// TIA Portal V20 export
FUNCTION_BLOCK "Sequence_2_TransferPnPRight"   // FB32855, LAD
TITLE = Sequence
// Sequence template programmend in ladder logic
// stored: IsIECCheckEnabled true, MemoryReserve 100, Namespace Unit1.Em5, SetENOAutomatically true
   VAR_INPUT
      unitStatus { ExternalAccessible := 'False'; ExternalVisible := 'False'; ExternalWritable := 'False'} : "LAF_typeUnitStatus";
   END_VAR
   VAR
      instSequenceLADControl { ExternalAccessible := 'False'; ExternalVisible := 'False'; ExternalWritable := 'False'} : "LAF_ControlLadSequence";
      instSequenceLADStatus { ExternalAccessible := 'False'; ExternalVisible := 'False'; ExternalWritable := 'False'} : "LAF_StatusLadSequence";
      statTonTime { ExternalAccessible := 'False'; ExternalVisible := 'False'; ExternalWritable := 'False'} : Array[0..9999] of TON_TIME;
      NoDataCheck { S7_SetPoint := 'True'} : "LER_typePartData";
   END_VAR
   VAR_TEMP
      tempCustomerAction : Bool;   // Placeholder for possible actions
      tempDo_nothing_and_wait_for_init : Bool;   // Placeholder for doing nothing
      tempSafeStateCondition : Bool;   // Temp Condition for the equipment module to be in a safe state
   END_VAR
   VAR CONSTANT
      delayTime : Time := T#500ms;
      STEP_IDLE : DInt := 1;
      JOB_1_STEP_01 : DInt := 101;
      JOB_1_STEP_10 : DInt := 110;
      JOB_1_STEP_20 : DInt := 120;
      JOB_1_STEP_30 : DInt := 130;
      JOB_1_STEP_40 : DInt := 140;
      JOB_1_STEP_50 : DInt := 150;
      JOB_1_STEP_60 : DInt := 160;
      JOB_1_STEP_70 : DInt := 170;
      JOB_1_STEP_80 : DInt := 180;
      JOB_1_STEP_90 : DInt := 190;
      JOB_2_STEP_01 : DInt := 201;
      JOB_2_STEP_10 : DInt := 210;
      JOB_2_STEP_20 : DInt := 220;
      JOB_2_STEP_30 : DInt := 230;
      JOB_2_STEP_40 : DInt := 240;
      JOB_2_STEP_80 : DInt := 280;
      JOB_2_STEP_81 : DInt := 281;
      JOB_2_STEP_90 : DInt := 290;
      JOB_3_STEP_01 : DInt := 301;
      JOB_3_STEP_10 : DInt := 310;
      JOB_3_STEP_20 : DInt := 320;
      JOB_3_STEP_30 : DInt := 330;
      JOB_3_STEP_40 : DInt := 340;
      JOB_3_STEP_50 : DInt := 350;
      JOB_3_STEP_80 : DInt := 380;
      JOB_3_STEP_81 : DInt := 381;
      JOB_3_STEP_90 : DInt := 390;
      JOB_4_STEP_01 : DInt := 401;
      JOB_4_STEP_10 : DInt := 410;
      JOB_4_STEP_20 : DInt := 420;
      JOB_4_STEP_30 : DInt := 430;
      JOB_4_STEP_40 : DInt := 440;
      JOB_4_STEP_80 : DInt := 480;
      JOB_4_STEP_81 : DInt := 481;
      JOB_4_STEP_90 : DInt := 490;
      JOB_5_STEP_01 : DInt := 501;
      JOB_5_STEP_10 : DInt := 510;
      JOB_5_STEP_20 : DInt := 520;
      JOB_5_STEP_30 : DInt := 530;
      JOB_5_STEP_40 : DInt := 540;
      JOB_5_STEP_50 : DInt := 550;
      JOB_5_STEP_80 : DInt := 580;
      JOB_5_STEP_81 : DInt := 581;
      JOB_5_STEP_90 : DInt := 590;
      JOB_6_STEP_01 : DInt := 601;
      JOB_6_STEP_10 : DInt := 610;
      JOB_6_STEP_20 : DInt := 620;
      JOB_6_STEP_30 : DInt := 630;
      JOB_6_STEP_40 : DInt := 640;
      JOB_6_STEP_50 : DInt := 650;
      JOB_6_STEP_51 : DInt := 651;
      JOB_6_STEP_52 : DInt := 652;
      JOB_6_STEP_80 : DInt := 680;
      JOB_6_STEP_81 : DInt := 681;
      JOB_6_STEP_90 : DInt := 690;
      JOB_7_STEP_01 : DInt := 701;
      JOB_7_STEP_10 : DInt := 710;
      JOB_7_STEP_20 : DInt := 720;
      JOB_7_STEP_30 : DInt := 730;
      JOB_7_STEP_40 : DInt := 740;
      JOB_7_STEP_50 : DInt := 750;
      JOB_7_STEP_80 : DInt := 780;
      JOB_7_STEP_81 : DInt := 781;
      JOB_7_STEP_90 : DInt := 790;
      JOB_8_STEP_01 : DInt := 801;
      JOB_8_STEP_10 : DInt := 810;
      JOB_8_STEP_20 : DInt := 820;
      JOB_8_STEP_30 : DInt := 830;
      JOB_8_STEP_40 : DInt := 840;
      JOB_8_STEP_50 : DInt := 850;
      JOB_8_STEP_51 : DInt := 851;
      JOB_8_STEP_52 : DInt := 852;
      JOB_8_STEP_80 : DInt := 880;
      JOB_8_STEP_81 : DInt := 881;
      JOB_8_STEP_90 : DInt := 890;
      JOB_9_STEP_01 : DInt := 901;
      JOB_9_STEP_10 : DInt := 910;
      JOB_9_STEP_20 : DInt := 920;
      JOB_9_STEP_30 : DInt := 930;
      JOB_9_STEP_31 : DInt := 931;
      JOB_9_STEP_40 : DInt := 940;
      JOB_9_STEP_50 : DInt := 950;
      JOB_9_STEP_80 : DInt := 980;
      JOB_9_STEP_81 : DInt := 981;
      JOB_9_STEP_82 : DInt := 982;
      JOB_9_STEP_90 : DInt := 990;
      STEP_IMMEDIATE_STOP : DInt := 9001;   // Step executed when an immediate stop command is triggered for the sequence (i.e. when unit is in state aborting)
      TO_DO_INSERT_ACTIONS_HERE : Bool := TRUE;   // Template : Add actions
      TO_DO_INSERT_CONDITION_FOR_TRANSITION_HERE : Bool := TRUE;   // Template : Add conditions
   END_VAR
   VAR_TEMP   // added for the SCL form of the ladder/FBD networks
      _w1 : Bool;
      _w2 : Bool;
      _w3 : Bool;
      _w4 : Bool;
      _w5 : Bool;
      _w6 : Bool;
   END_VAR
BEGIN

REGION Network 1: BLOCK INFO HEADER
   // (company) / (C) Copyright (year)
   // ---------------------------------------------------------------------------------
   // Title:                             (Title of this block)
   // Comment/Function: (that is implemented in the block)
   // Library/Family:           (that the source is dedicated to)
   // Author:                        (department / person in charge / contact)
   // Target System:          (test system with FW version)
   // Engineering:              TIA Portal (SW version)
   // Restrictions:               (OB types, etc.)
   // Requirements:           (hardware, technological package, etc.)
   // ---------------------------------------------------------------------------------
   // Change log table:
   // Version          | Date             | Signature      | Expert in charge  | Changes applied ------------------------|----------------------|-------------------------|--------------------------------|-----------------------
   // 001.000.000 | yyyy-mm-dd | 0x00000000 | (name of expert) | First released version
END_REGION

REGION Network 2: DESCRIPTION
   // This is a template block provided by the Automation Framework. It can be used to create an own project.
   // The Block Info Header is prepared to put in your own data.
   // Description of the block could be added here and the docu created by Code2Docu.
END_REGION

REGION Network 3: ********************* CONTROL *************************
END_REGION

REGION Network 4: Sequence Control ("Enter your Sequins number here")
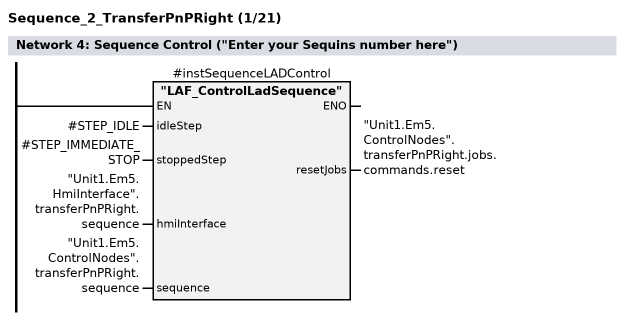
   RUNG wire#powerrail
      #instSequenceLADControl(idleStep := #STEP_IDLE, stoppedStep := #STEP_IMMEDIATE_STOP, hmiInterface := "Unit1.Em5.HmiInterface".transferPnPRight.sequence, sequence := "Unit1.Em5.ControlNodes".transferPnPRight.sequence, resetJobs => "Unit1.Em5.ControlNodes".transferPnPRight.jobs.commands.reset)
   END_RUNG
   // the same network as SCL:
   #instSequenceLADControl(idleStep := #STEP_IDLE,   // "LAF_ControlLadSequence"
                           stoppedStep := #STEP_IMMEDIATE_STOP,
                           hmiInterface := "Unit1.Em5.HmiInterface".transferPnPRight.sequence,
                           sequence := "Unit1.Em5.ControlNodes".transferPnPRight.sequence,
                           resetJobs => "Unit1.Em5.ControlNodes".transferPnPRight.jobs.commands.reset);
END_REGION

REGION Network 5: Step Idle
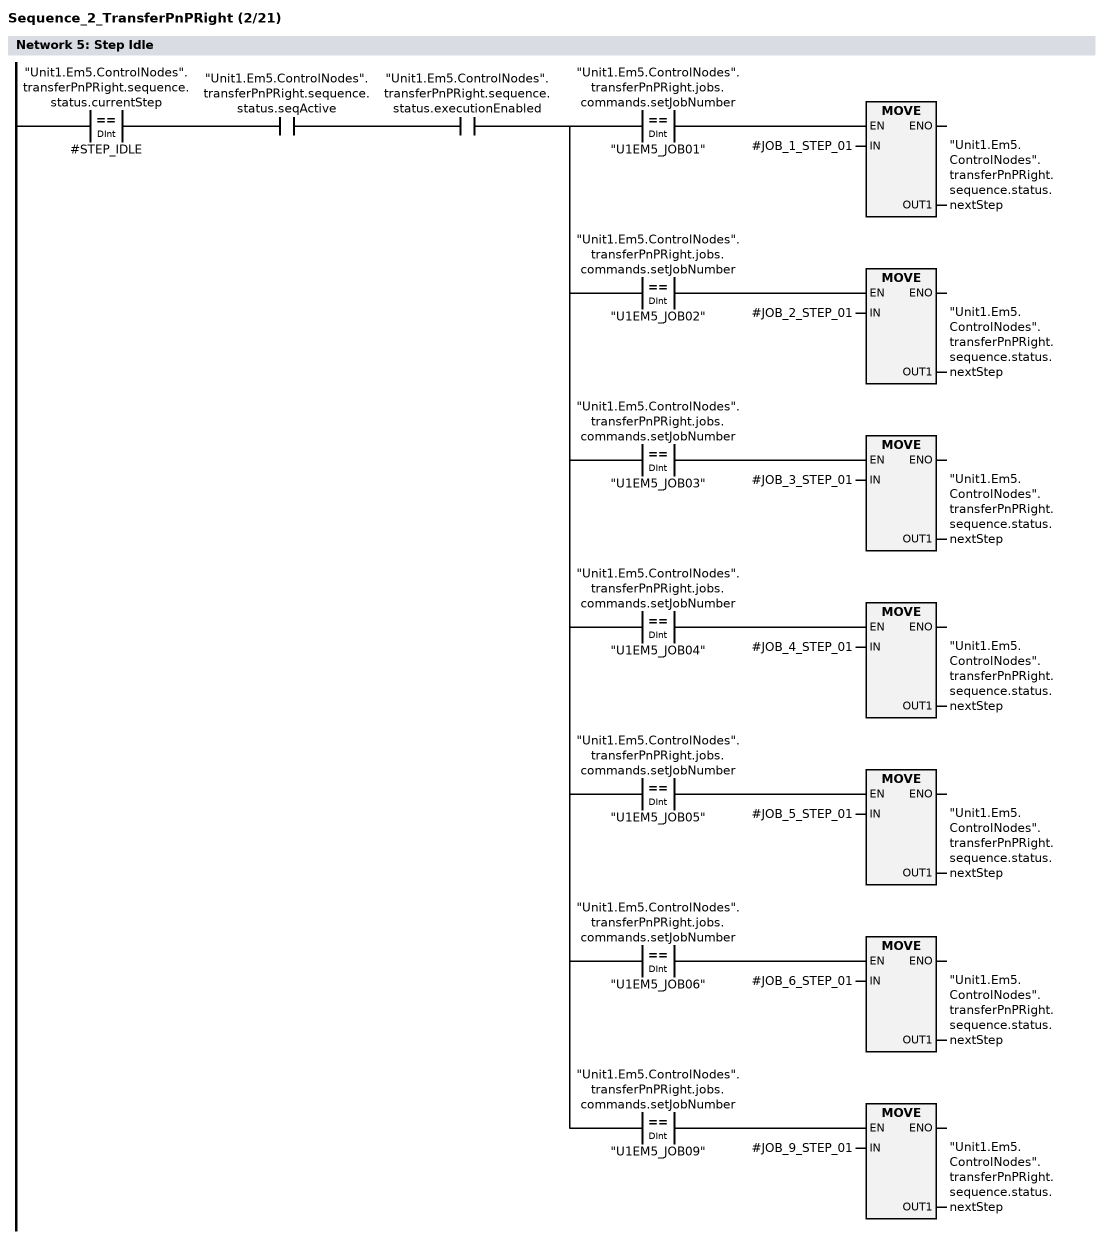
   RUNG wire#powerrail
      { S7_Templates := "SrcType := DInt" } EQ_Contact(in1 := "Unit1.Em5.ControlNodes".transferPnPRight.sequence.status.currentStep, in2 := #STEP_IDLE)
      Contact( "Unit1.Em5.ControlNodes".transferPnPRight.sequence.status.seqActive )
      Contact( "Unit1.Em5.ControlNodes".transferPnPRight.sequence.status.executionEnabled )
      wire#w1
      { S7_Templates := "SrcType := DInt" } EQ_Contact(in1 := "Unit1.Em5.ControlNodes".transferPnPRight.jobs.commands.setJobNumber, in2 := "U1EM5_JOB01")
      Move(in := #JOB_1_STEP_01, out1 => "Unit1.Em5.ControlNodes".transferPnPRight.sequence.status.nextStep)
   END_RUNG
   RUNG wire#w1
      { S7_Templates := "SrcType := DInt" } EQ_Contact(in1 := "Unit1.Em5.ControlNodes".transferPnPRight.jobs.commands.setJobNumber, in2 := "U1EM5_JOB02")
      Move(in := #JOB_2_STEP_01, out1 => "Unit1.Em5.ControlNodes".transferPnPRight.sequence.status.nextStep)
   END_RUNG
   RUNG wire#w1
      { S7_Templates := "SrcType := DInt" } EQ_Contact(in1 := "Unit1.Em5.ControlNodes".transferPnPRight.jobs.commands.setJobNumber, in2 := "U1EM5_JOB03")
      Move(in := #JOB_3_STEP_01, out1 => "Unit1.Em5.ControlNodes".transferPnPRight.sequence.status.nextStep)
   END_RUNG
   RUNG wire#w1
      { S7_Templates := "SrcType := DInt" } EQ_Contact(in1 := "Unit1.Em5.ControlNodes".transferPnPRight.jobs.commands.setJobNumber, in2 := "U1EM5_JOB04")
      Move(in := #JOB_4_STEP_01, out1 => "Unit1.Em5.ControlNodes".transferPnPRight.sequence.status.nextStep)
   END_RUNG
   RUNG wire#w1
      { S7_Templates := "SrcType := DInt" } EQ_Contact(in1 := "Unit1.Em5.ControlNodes".transferPnPRight.jobs.commands.setJobNumber, in2 := "U1EM5_JOB05")
      Move(in := #JOB_5_STEP_01, out1 => "Unit1.Em5.ControlNodes".transferPnPRight.sequence.status.nextStep)
   END_RUNG
   RUNG wire#w1
      { S7_Templates := "SrcType := DInt" } EQ_Contact(in1 := "Unit1.Em5.ControlNodes".transferPnPRight.jobs.commands.setJobNumber, in2 := "U1EM5_JOB06")
      Move(in := #JOB_6_STEP_01, out1 => "Unit1.Em5.ControlNodes".transferPnPRight.sequence.status.nextStep)
   END_RUNG
   RUNG wire#w1
      { S7_Templates := "SrcType := DInt" } EQ_Contact(in1 := "Unit1.Em5.ControlNodes".transferPnPRight.jobs.commands.setJobNumber, in2 := "U1EM5_JOB09")
      Move(in := #JOB_9_STEP_01, out1 => "Unit1.Em5.ControlNodes".transferPnPRight.sequence.status.nextStep)
   END_RUNG
   // the same network as SCL:
   #_w1 := ("Unit1.Em5.ControlNodes".transferPnPRight.sequence.status.currentStep = #STEP_IDLE) AND "Unit1.Em5.ControlNodes".transferPnPRight.sequence.status.seqActive AND "Unit1.Em5.ControlNodes".transferPnPRight.sequence.status.executionEnabled;
   IF #_w1 AND ("Unit1.Em5.ControlNodes".transferPnPRight.jobs.commands.setJobNumber = "U1EM5_JOB01") THEN
       "Unit1.Em5.ControlNodes".transferPnPRight.sequence.status.nextStep := #JOB_1_STEP_01;
   END_IF;
   IF #_w1 AND ("Unit1.Em5.ControlNodes".transferPnPRight.jobs.commands.setJobNumber = "U1EM5_JOB02") THEN
       "Unit1.Em5.ControlNodes".transferPnPRight.sequence.status.nextStep := #JOB_2_STEP_01;
   END_IF;
   IF #_w1 AND ("Unit1.Em5.ControlNodes".transferPnPRight.jobs.commands.setJobNumber = "U1EM5_JOB03") THEN
       "Unit1.Em5.ControlNodes".transferPnPRight.sequence.status.nextStep := #JOB_3_STEP_01;
   END_IF;
   IF #_w1 AND ("Unit1.Em5.ControlNodes".transferPnPRight.jobs.commands.setJobNumber = "U1EM5_JOB04") THEN
       "Unit1.Em5.ControlNodes".transferPnPRight.sequence.status.nextStep := #JOB_4_STEP_01;
   END_IF;
   IF #_w1 AND ("Unit1.Em5.ControlNodes".transferPnPRight.jobs.commands.setJobNumber = "U1EM5_JOB05") THEN
       "Unit1.Em5.ControlNodes".transferPnPRight.sequence.status.nextStep := #JOB_5_STEP_01;
   END_IF;
   IF #_w1 AND ("Unit1.Em5.ControlNodes".transferPnPRight.jobs.commands.setJobNumber = "U1EM5_JOB06") THEN
       "Unit1.Em5.ControlNodes".transferPnPRight.sequence.status.nextStep := #JOB_6_STEP_01;
   END_IF;
   IF #_w1 AND ("Unit1.Em5.ControlNodes".transferPnPRight.jobs.commands.setJobNumber = "U1EM5_JOB09") THEN
       "Unit1.Em5.ControlNodes".transferPnPRight.sequence.status.nextStep := #JOB_9_STEP_01;
   END_IF;
END_REGION

REGION Network 6: *************** JOB[1] EM HOMING ************************
END_REGION

REGION Network 7: Step[101] : JOB[1] Condition
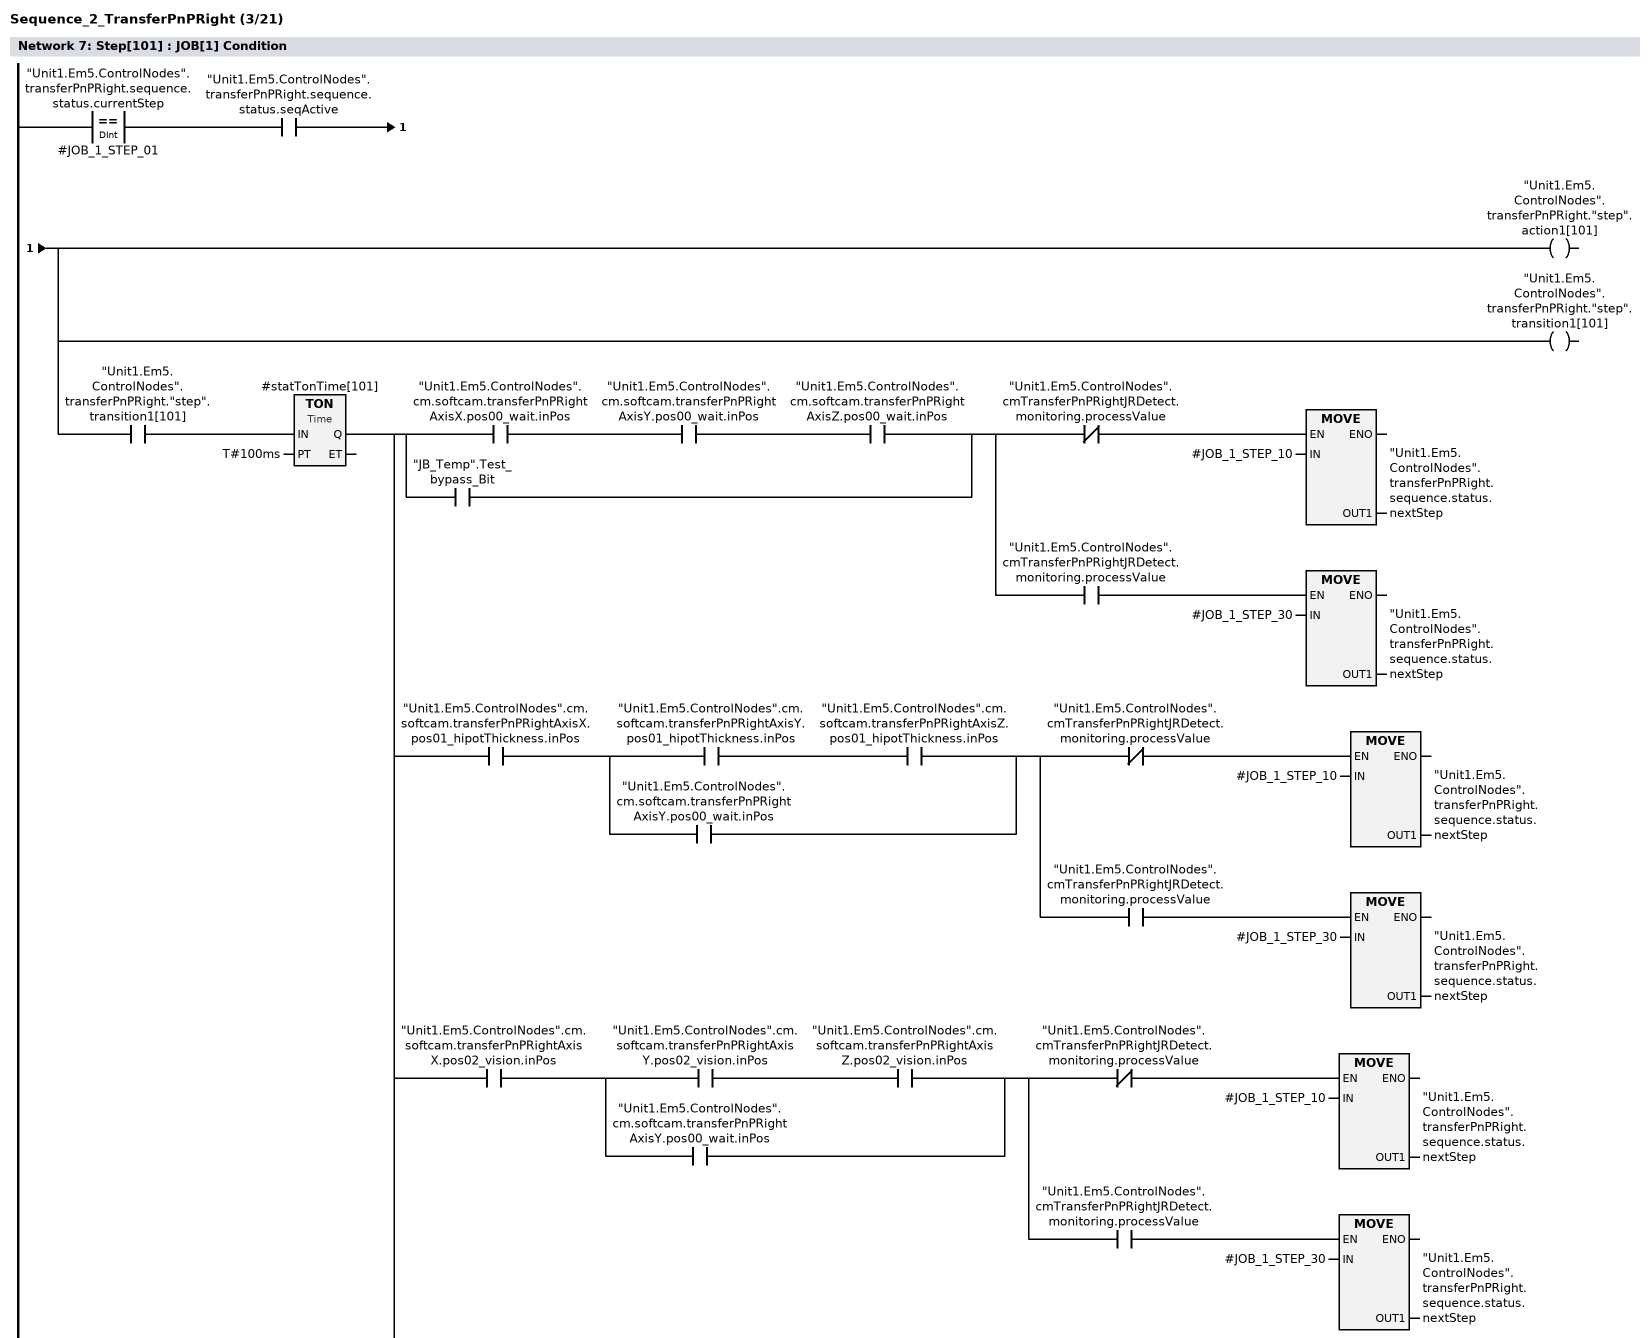
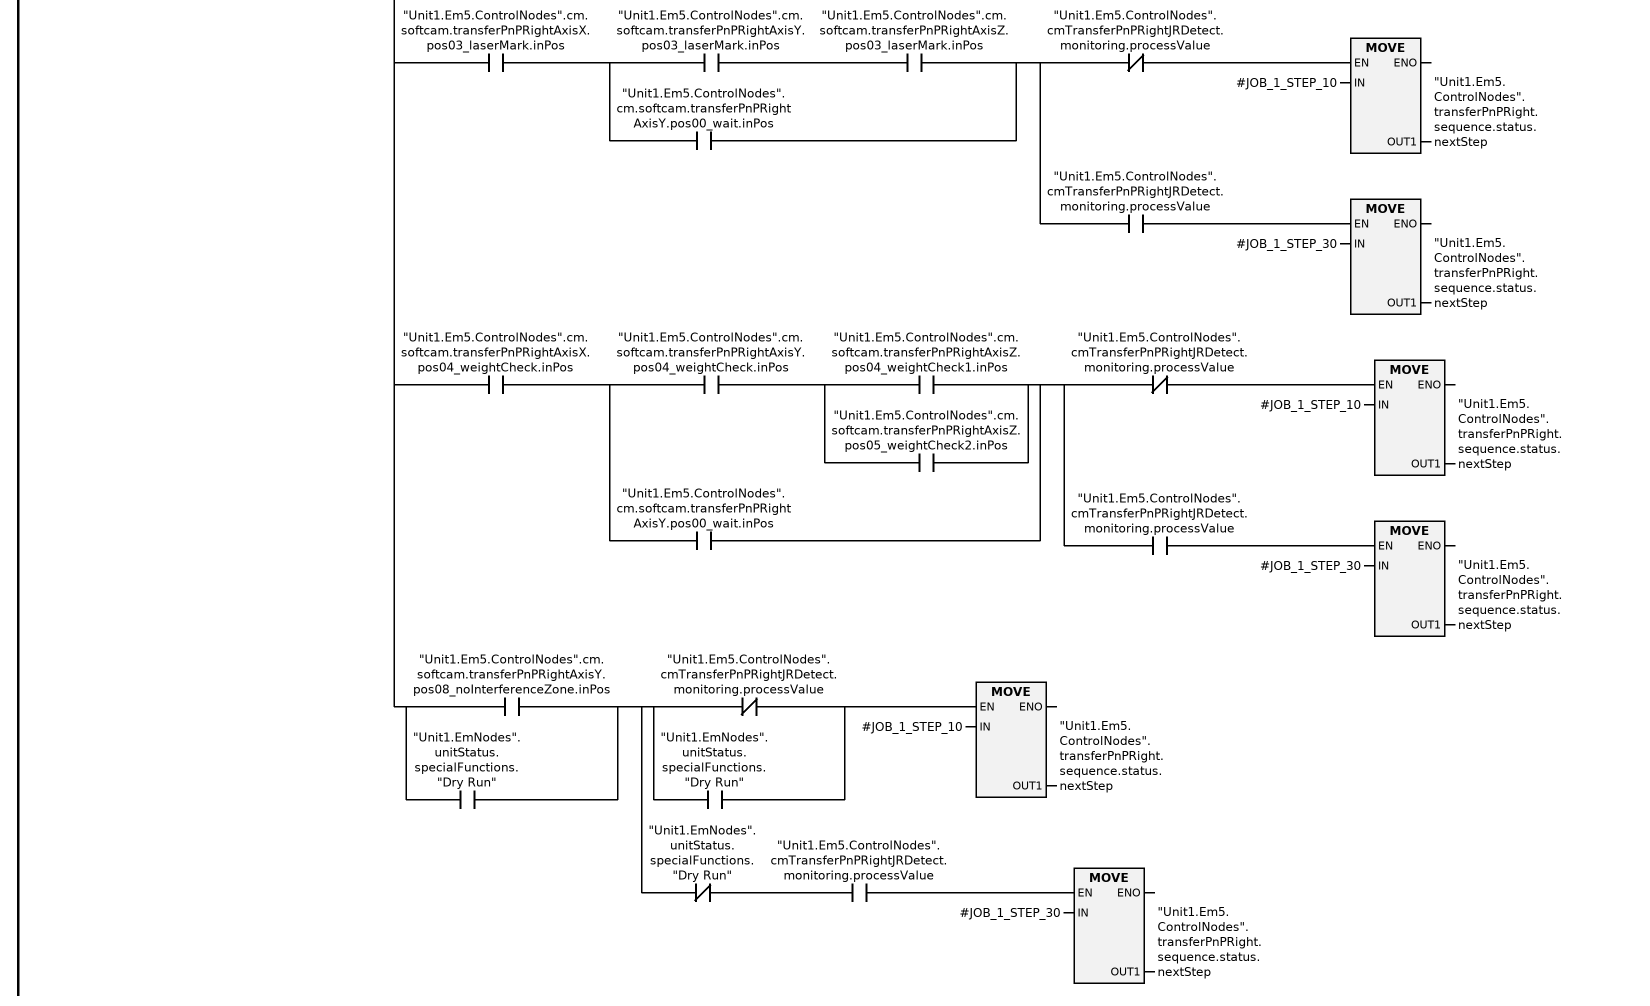
   RUNG wire#powerrail
      { S7_Templates := "SrcType := DInt" } EQ_Contact(in1 := "Unit1.Em5.ControlNodes".transferPnPRight.sequence.status.currentStep, in2 := #JOB_1_STEP_01)
      Contact( "Unit1.Em5.ControlNodes".transferPnPRight.sequence.status.seqActive )
      wire#w1
      Coil( "Unit1.Em5.ControlNodes".transferPnPRight."step".action1[101] )
   END_RUNG
   RUNG wire#w1
      Coil( "Unit1.Em5.ControlNodes".transferPnPRight."step".transition1[101] )
   END_RUNG
   RUNG wire#w1
      Contact( "Unit1.Em5.ControlNodes".transferPnPRight."step".transition1[101] )
      { S7_Templates := "time_type := Time" } #statTonTime[101].TON(pt := T#100ms, et =>)
      wire#w2
      Contact( "Unit1.Em5.ControlNodes".cm.softcam.transferPnPRightAxisX.pos00_wait.inPos )
      Contact( "Unit1.Em5.ControlNodes".cm.softcam.transferPnPRightAxisY.pos00_wait.inPos )
      Contact( "Unit1.Em5.ControlNodes".cm.softcam.transferPnPRightAxisZ.pos00_wait.inPos )
      wire#w3
      I_Contact( "Unit1.Em5.ControlNodes".cmTransferPnPRightJRDetect.monitoring.processValue )
      Move(in := #JOB_1_STEP_10, out1 => "Unit1.Em5.ControlNodes".transferPnPRight.sequence.status.nextStep)
   END_RUNG
   RUNG wire#w2
      Contact( "JB_Temp".Test_bypass_Bit )
   END_RUNG wire#w3
   RUNG wire#w3
      Contact( "Unit1.Em5.ControlNodes".cmTransferPnPRightJRDetect.monitoring.processValue )
      Move(in := #JOB_1_STEP_30, out1 => "Unit1.Em5.ControlNodes".transferPnPRight.sequence.status.nextStep)
   END_RUNG
   RUNG wire#w2
      Contact( "Unit1.Em5.ControlNodes".cm.softcam.transferPnPRightAxisX.pos01_hipotThickness.inPos )
      wire#w4
      Contact( "Unit1.Em5.ControlNodes".cm.softcam.transferPnPRightAxisY.pos01_hipotThickness.inPos )
      Contact( "Unit1.Em5.ControlNodes".cm.softcam.transferPnPRightAxisZ.pos01_hipotThickness.inPos )
      wire#w5
      I_Contact( "Unit1.Em5.ControlNodes".cmTransferPnPRightJRDetect.monitoring.processValue )
      Move(in := #JOB_1_STEP_10, out1 => "Unit1.Em5.ControlNodes".transferPnPRight.sequence.status.nextStep)
   END_RUNG
   RUNG wire#w4
      Contact( "Unit1.Em5.ControlNodes".cm.softcam.transferPnPRightAxisY.pos00_wait.inPos )
   END_RUNG wire#w5
   RUNG wire#w5
      Contact( "Unit1.Em5.ControlNodes".cmTransferPnPRightJRDetect.monitoring.processValue )
      Move(in := #JOB_1_STEP_30, out1 => "Unit1.Em5.ControlNodes".transferPnPRight.sequence.status.nextStep)
   END_RUNG
   RUNG wire#w2
      Contact( "Unit1.Em5.ControlNodes".cm.softcam.transferPnPRightAxisX.pos02_vision.inPos )
      wire#w6
      Contact( "Unit1.Em5.ControlNodes".cm.softcam.transferPnPRightAxisY.pos02_vision.inPos )
      Contact( "Unit1.Em5.ControlNodes".cm.softcam.transferPnPRightAxisZ.pos02_vision.inPos )
      wire#w7
      I_Contact( "Unit1.Em5.ControlNodes".cmTransferPnPRightJRDetect.monitoring.processValue )
      Move(in := #JOB_1_STEP_10, out1 => "Unit1.Em5.ControlNodes".transferPnPRight.sequence.status.nextStep)
   END_RUNG
   RUNG wire#w6
      Contact( "Unit1.Em5.ControlNodes".cm.softcam.transferPnPRightAxisY.pos00_wait.inPos )
   END_RUNG wire#w7
   RUNG wire#w7
      Contact( "Unit1.Em5.ControlNodes".cmTransferPnPRightJRDetect.monitoring.processValue )
      Move(in := #JOB_1_STEP_30, out1 => "Unit1.Em5.ControlNodes".transferPnPRight.sequence.status.nextStep)
   END_RUNG
   RUNG wire#w2
      Contact( "Unit1.Em5.ControlNodes".cm.softcam.transferPnPRightAxisX.pos03_laserMark.inPos )
      wire#w8
      Contact( "Unit1.Em5.ControlNodes".cm.softcam.transferPnPRightAxisY.pos03_laserMark.inPos )
      Contact( "Unit1.Em5.ControlNodes".cm.softcam.transferPnPRightAxisZ.pos03_laserMark.inPos )
      wire#w9
      I_Contact( "Unit1.Em5.ControlNodes".cmTransferPnPRightJRDetect.monitoring.processValue )
      Move(in := #JOB_1_STEP_10, out1 => "Unit1.Em5.ControlNodes".transferPnPRight.sequence.status.nextStep)
   END_RUNG
   RUNG wire#w8
      Contact( "Unit1.Em5.ControlNodes".cm.softcam.transferPnPRightAxisY.pos00_wait.inPos )
   END_RUNG wire#w9
   RUNG wire#w9
      Contact( "Unit1.Em5.ControlNodes".cmTransferPnPRightJRDetect.monitoring.processValue )
      Move(in := #JOB_1_STEP_30, out1 => "Unit1.Em5.ControlNodes".transferPnPRight.sequence.status.nextStep)
   END_RUNG
   RUNG wire#w2
      Contact( "Unit1.Em5.ControlNodes".cm.softcam.transferPnPRightAxisX.pos04_weightCheck.inPos )
      wire#w10
      Contact( "Unit1.Em5.ControlNodes".cm.softcam.transferPnPRightAxisY.pos04_weightCheck.inPos )
      wire#w11
      Contact( "Unit1.Em5.ControlNodes".cm.softcam.transferPnPRightAxisZ.pos04_weightCheck1.inPos )
      wire#w12
      I_Contact( "Unit1.Em5.ControlNodes".cmTransferPnPRightJRDetect.monitoring.processValue )
      Move(in := #JOB_1_STEP_10, out1 => "Unit1.Em5.ControlNodes".transferPnPRight.sequence.status.nextStep)
   END_RUNG
   RUNG wire#w11
      Contact( "Unit1.Em5.ControlNodes".cm.softcam.transferPnPRightAxisZ.pos05_weightCheck2.inPos )
   END_RUNG wire#w12
   RUNG wire#w10
      Contact( "Unit1.Em5.ControlNodes".cm.softcam.transferPnPRightAxisY.pos00_wait.inPos )
   END_RUNG wire#w12
   RUNG wire#w12
      Contact( "Unit1.Em5.ControlNodes".cmTransferPnPRightJRDetect.monitoring.processValue )
      Move(in := #JOB_1_STEP_30, out1 => "Unit1.Em5.ControlNodes".transferPnPRight.sequence.status.nextStep)
   END_RUNG
   RUNG wire#w2
      Contact( "Unit1.Em5.ControlNodes".cm.softcam.transferPnPRightAxisY.pos08_noInterferenceZone.inPos )
      wire#w13
      I_Contact( "Unit1.Em5.ControlNodes".cmTransferPnPRightJRDetect.monitoring.processValue )
      wire#w14
      Move(in := #JOB_1_STEP_10, out1 => "Unit1.Em5.ControlNodes".transferPnPRight.sequence.status.nextStep)
   END_RUNG
   RUNG wire#w2
      Contact( "Unit1.EmNodes".unitStatus.specialFunctions."Dry Run" )
   END_RUNG wire#w13
   RUNG wire#w13
      Contact( "Unit1.EmNodes".unitStatus.specialFunctions."Dry Run" )
   END_RUNG wire#w14
   RUNG wire#w13
      I_Contact( "Unit1.EmNodes".unitStatus.specialFunctions."Dry Run" )
      Contact( "Unit1.Em5.ControlNodes".cmTransferPnPRightJRDetect.monitoring.processValue )
      Move(in := #JOB_1_STEP_30, out1 => "Unit1.Em5.ControlNodes".transferPnPRight.sequence.status.nextStep)
   END_RUNG
   // the same network as SCL:
   "Unit1.Em5.ControlNodes".transferPnPRight."step".action1[101] := ("Unit1.Em5.ControlNodes".transferPnPRight.sequence.status.currentStep = #JOB_1_STEP_01) AND "Unit1.Em5.ControlNodes".transferPnPRight.sequence.status.seqActive;
   "Unit1.Em5.ControlNodes".transferPnPRight."step".transition1[101] := ("Unit1.Em5.ControlNodes".transferPnPRight.sequence.status.currentStep = #JOB_1_STEP_01) AND "Unit1.Em5.ControlNodes".transferPnPRight.sequence.status.seqActive;
   #statTonTime[101].TON(IN := ("Unit1.Em5.ControlNodes".transferPnPRight.sequence.status.currentStep = #JOB_1_STEP_01) AND "Unit1.Em5.ControlNodes".transferPnPRight.sequence.status.seqActive AND "Unit1.Em5.ControlNodes".transferPnPRight."step".transition1[101],
                         PT := T#100ms);
   #_w1 := #statTonTime[101].Q AND (("Unit1.Em5.ControlNodes".cm.softcam.transferPnPRightAxisX.pos00_wait.inPos AND "Unit1.Em5.ControlNodes".cm.softcam.transferPnPRightAxisY.pos00_wait.inPos AND "Unit1.Em5.ControlNodes".cm.softcam.transferPnPRightAxisZ.pos00_wait.inPos) OR "JB_Temp".Test_bypass_Bit);
   IF #_w1 AND NOT "Unit1.Em5.ControlNodes".cmTransferPnPRightJRDetect.monitoring.processValue THEN
       "Unit1.Em5.ControlNodes".transferPnPRight.sequence.status.nextStep := #JOB_1_STEP_10;
   END_IF;
   IF #_w1 AND "Unit1.Em5.ControlNodes".cmTransferPnPRightJRDetect.monitoring.processValue THEN
       "Unit1.Em5.ControlNodes".transferPnPRight.sequence.status.nextStep := #JOB_1_STEP_30;
   END_IF;
   #_w2 := #statTonTime[101].Q AND "Unit1.Em5.ControlNodes".cm.softcam.transferPnPRightAxisX.pos01_hipotThickness.inPos AND (("Unit1.Em5.ControlNodes".cm.softcam.transferPnPRightAxisY.pos01_hipotThickness.inPos AND "Unit1.Em5.ControlNodes".cm.softcam.transferPnPRightAxisZ.pos01_hipotThickness.inPos) OR "Unit1.Em5.ControlNodes".cm.softcam.transferPnPRightAxisY.pos00_wait.inPos);
   IF #_w2 AND NOT "Unit1.Em5.ControlNodes".cmTransferPnPRightJRDetect.monitoring.processValue THEN
       "Unit1.Em5.ControlNodes".transferPnPRight.sequence.status.nextStep := #JOB_1_STEP_10;
   END_IF;
   IF #_w2 AND "Unit1.Em5.ControlNodes".cmTransferPnPRightJRDetect.monitoring.processValue THEN
       "Unit1.Em5.ControlNodes".transferPnPRight.sequence.status.nextStep := #JOB_1_STEP_30;
   END_IF;
   #_w3 := #statTonTime[101].Q AND "Unit1.Em5.ControlNodes".cm.softcam.transferPnPRightAxisX.pos02_vision.inPos AND (("Unit1.Em5.ControlNodes".cm.softcam.transferPnPRightAxisY.pos02_vision.inPos AND "Unit1.Em5.ControlNodes".cm.softcam.transferPnPRightAxisZ.pos02_vision.inPos) OR "Unit1.Em5.ControlNodes".cm.softcam.transferPnPRightAxisY.pos00_wait.inPos);
   IF #_w3 AND NOT "Unit1.Em5.ControlNodes".cmTransferPnPRightJRDetect.monitoring.processValue THEN
       "Unit1.Em5.ControlNodes".transferPnPRight.sequence.status.nextStep := #JOB_1_STEP_10;
   END_IF;
   IF #_w3 AND "Unit1.Em5.ControlNodes".cmTransferPnPRightJRDetect.monitoring.processValue THEN
       "Unit1.Em5.ControlNodes".transferPnPRight.sequence.status.nextStep := #JOB_1_STEP_30;
   END_IF;
   #_w4 := #statTonTime[101].Q AND "Unit1.Em5.ControlNodes".cm.softcam.transferPnPRightAxisX.pos03_laserMark.inPos AND (("Unit1.Em5.ControlNodes".cm.softcam.transferPnPRightAxisY.pos03_laserMark.inPos AND "Unit1.Em5.ControlNodes".cm.softcam.transferPnPRightAxisZ.pos03_laserMark.inPos) OR "Unit1.Em5.ControlNodes".cm.softcam.transferPnPRightAxisY.pos00_wait.inPos);
   IF #_w4 AND NOT "Unit1.Em5.ControlNodes".cmTransferPnPRightJRDetect.monitoring.processValue THEN
       "Unit1.Em5.ControlNodes".transferPnPRight.sequence.status.nextStep := #JOB_1_STEP_10;
   END_IF;
   IF #_w4 AND "Unit1.Em5.ControlNodes".cmTransferPnPRightJRDetect.monitoring.processValue THEN
       "Unit1.Em5.ControlNodes".transferPnPRight.sequence.status.nextStep := #JOB_1_STEP_30;
   END_IF;
   #_w5 := #statTonTime[101].Q AND "Unit1.Em5.ControlNodes".cm.softcam.transferPnPRightAxisX.pos04_weightCheck.inPos AND (("Unit1.Em5.ControlNodes".cm.softcam.transferPnPRightAxisY.pos04_weightCheck.inPos AND ("Unit1.Em5.ControlNodes".cm.softcam.transferPnPRightAxisZ.pos04_weightCheck1.inPos OR "Unit1.Em5.ControlNodes".cm.softcam.transferPnPRightAxisZ.pos05_weightCheck2.inPos)) OR "Unit1.Em5.ControlNodes".cm.softcam.transferPnPRightAxisY.pos00_wait.inPos);
   IF #_w5 AND NOT "Unit1.Em5.ControlNodes".cmTransferPnPRightJRDetect.monitoring.processValue THEN
       "Unit1.Em5.ControlNodes".transferPnPRight.sequence.status.nextStep := #JOB_1_STEP_10;
   END_IF;
   IF #_w5 AND "Unit1.Em5.ControlNodes".cmTransferPnPRightJRDetect.monitoring.processValue THEN
       "Unit1.Em5.ControlNodes".transferPnPRight.sequence.status.nextStep := #JOB_1_STEP_30;
   END_IF;
   #_w6 := #statTonTime[101].Q AND ("Unit1.Em5.ControlNodes".cm.softcam.transferPnPRightAxisY.pos08_noInterferenceZone.inPos OR "Unit1.EmNodes".unitStatus.specialFunctions."Dry Run");
   IF #_w6 AND (NOT "Unit1.Em5.ControlNodes".cmTransferPnPRightJRDetect.monitoring.processValue OR "Unit1.EmNodes".unitStatus.specialFunctions."Dry Run") THEN
       "Unit1.Em5.ControlNodes".transferPnPRight.sequence.status.nextStep := #JOB_1_STEP_10;
   END_IF;
   IF #_w6 AND NOT "Unit1.EmNodes".unitStatus.specialFunctions."Dry Run" AND "Unit1.Em5.ControlNodes".cmTransferPnPRightJRDetect.monitoring.processValue THEN
       "Unit1.Em5.ControlNodes".transferPnPRight.sequence.status.nextStep := #JOB_1_STEP_30;
   END_IF;
END_REGION

REGION Network 8: Step[110] : Transfer PP Right Clamp Open
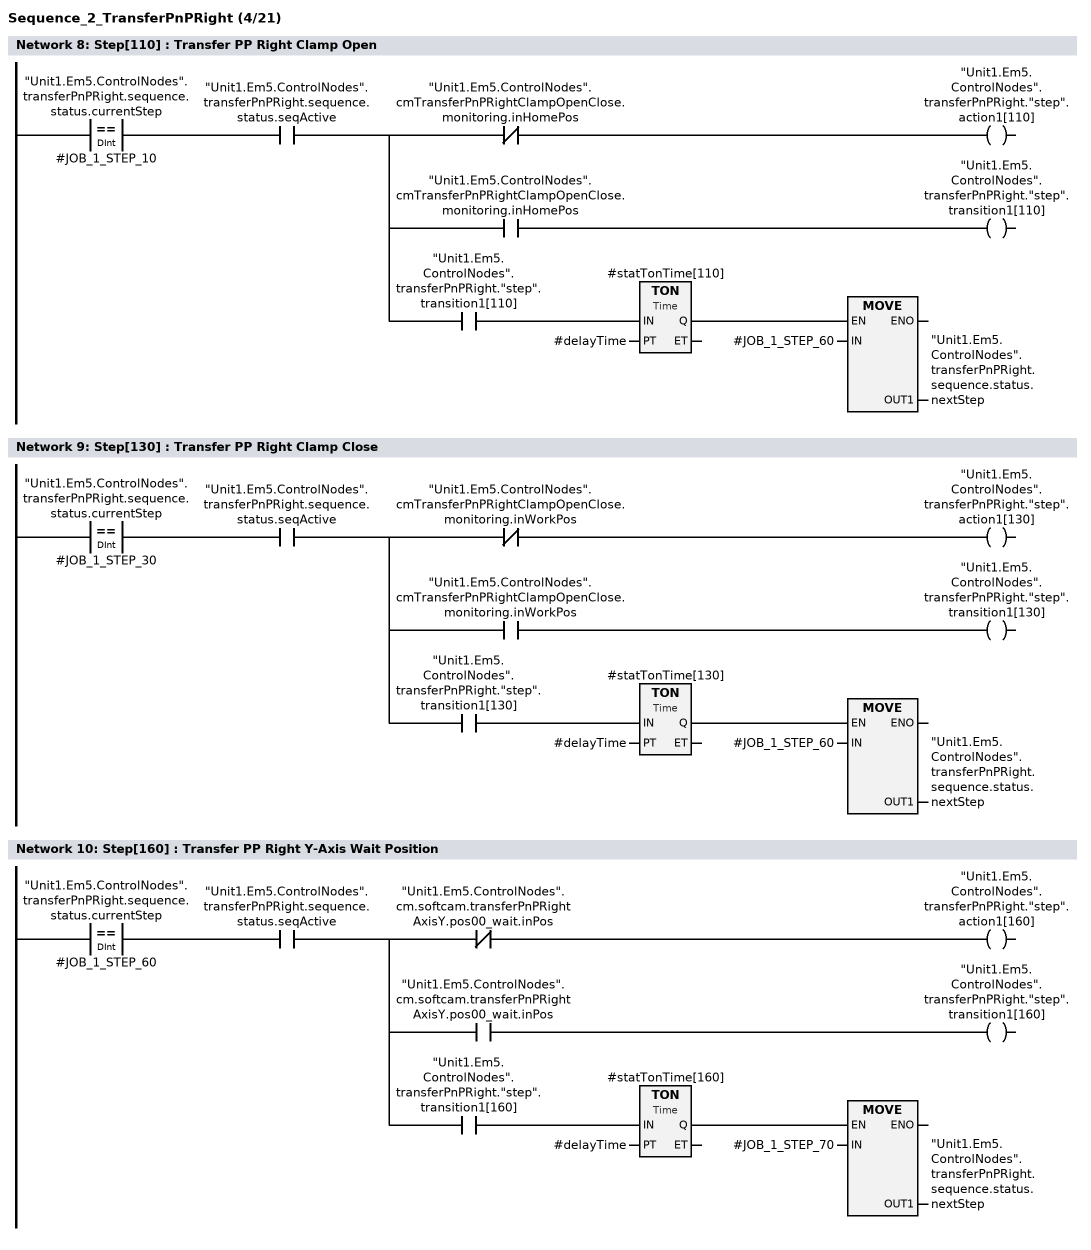
   RUNG wire#powerrail
      { S7_Templates := "SrcType := DInt" } EQ_Contact(in1 := "Unit1.Em5.ControlNodes".transferPnPRight.sequence.status.currentStep, in2 := #JOB_1_STEP_10)
      Contact( "Unit1.Em5.ControlNodes".transferPnPRight.sequence.status.seqActive )
      wire#w1
      I_Contact( "Unit1.Em5.ControlNodes".cmTransferPnPRightClampOpenClose.monitoring.inHomePos )
      Coil( "Unit1.Em5.ControlNodes".transferPnPRight."step".action1[110] )
   END_RUNG
   RUNG wire#w1
      Contact( "Unit1.Em5.ControlNodes".cmTransferPnPRightClampOpenClose.monitoring.inHomePos )
      Coil( "Unit1.Em5.ControlNodes".transferPnPRight."step".transition1[110] )
   END_RUNG
   RUNG wire#w1
      Contact( "Unit1.Em5.ControlNodes".transferPnPRight."step".transition1[110] )
      { S7_Templates := "time_type := Time" } #statTonTime[110].TON(pt := #delayTime, et =>)
      Move(in := #JOB_1_STEP_60, out1 => "Unit1.Em5.ControlNodes".transferPnPRight.sequence.status.nextStep)
   END_RUNG
   // the same network as SCL:
   #_w1 := ("Unit1.Em5.ControlNodes".transferPnPRight.sequence.status.currentStep = #JOB_1_STEP_10) AND "Unit1.Em5.ControlNodes".transferPnPRight.sequence.status.seqActive;
   "Unit1.Em5.ControlNodes".transferPnPRight."step".action1[110] := #_w1 AND NOT "Unit1.Em5.ControlNodes".cmTransferPnPRightClampOpenClose.monitoring.inHomePos;
   "Unit1.Em5.ControlNodes".transferPnPRight."step".transition1[110] := #_w1 AND "Unit1.Em5.ControlNodes".cmTransferPnPRightClampOpenClose.monitoring.inHomePos;
   #statTonTime[110].TON(IN := #_w1 AND "Unit1.Em5.ControlNodes".transferPnPRight."step".transition1[110],
                         PT := #delayTime);
   IF #statTonTime[110].Q THEN
       "Unit1.Em5.ControlNodes".transferPnPRight.sequence.status.nextStep := #JOB_1_STEP_60;
   END_IF;
END_REGION

REGION Network 9: Step[130] : Transfer PP Right Clamp Close
   RUNG wire#powerrail
      { S7_Templates := "SrcType := DInt" } EQ_Contact(in1 := "Unit1.Em5.ControlNodes".transferPnPRight.sequence.status.currentStep, in2 := #JOB_1_STEP_30)
      Contact( "Unit1.Em5.ControlNodes".transferPnPRight.sequence.status.seqActive )
      wire#w1
      I_Contact( "Unit1.Em5.ControlNodes".cmTransferPnPRightClampOpenClose.monitoring.inWorkPos )
      Coil( "Unit1.Em5.ControlNodes".transferPnPRight."step".action1[130] )
   END_RUNG
   RUNG wire#w1
      Contact( "Unit1.Em5.ControlNodes".cmTransferPnPRightClampOpenClose.monitoring.inWorkPos )
      Coil( "Unit1.Em5.ControlNodes".transferPnPRight."step".transition1[130] )
   END_RUNG
   RUNG wire#w1
      Contact( "Unit1.Em5.ControlNodes".transferPnPRight."step".transition1[130] )
      { S7_Templates := "time_type := Time" } #statTonTime[130].TON(pt := #delayTime, et =>)
      Move(in := #JOB_1_STEP_60, out1 => "Unit1.Em5.ControlNodes".transferPnPRight.sequence.status.nextStep)
   END_RUNG
   // the same network as SCL:
   #_w1 := ("Unit1.Em5.ControlNodes".transferPnPRight.sequence.status.currentStep = #JOB_1_STEP_30) AND "Unit1.Em5.ControlNodes".transferPnPRight.sequence.status.seqActive;
   "Unit1.Em5.ControlNodes".transferPnPRight."step".action1[130] := #_w1 AND NOT "Unit1.Em5.ControlNodes".cmTransferPnPRightClampOpenClose.monitoring.inWorkPos;
   "Unit1.Em5.ControlNodes".transferPnPRight."step".transition1[130] := #_w1 AND "Unit1.Em5.ControlNodes".cmTransferPnPRightClampOpenClose.monitoring.inWorkPos;
   #statTonTime[130].TON(IN := #_w1 AND "Unit1.Em5.ControlNodes".transferPnPRight."step".transition1[130],
                         PT := #delayTime);
   IF #statTonTime[130].Q THEN
       "Unit1.Em5.ControlNodes".transferPnPRight.sequence.status.nextStep := #JOB_1_STEP_60;
   END_IF;
END_REGION

REGION Network 10: Step[160] : Transfer PP Right Y-Axis Wait Position
   RUNG wire#powerrail
      { S7_Templates := "SrcType := DInt" } EQ_Contact(in1 := "Unit1.Em5.ControlNodes".transferPnPRight.sequence.status.currentStep, in2 := #JOB_1_STEP_60)
      Contact( "Unit1.Em5.ControlNodes".transferPnPRight.sequence.status.seqActive )
      wire#w1
      I_Contact( "Unit1.Em5.ControlNodes".cm.softcam.transferPnPRightAxisY.pos00_wait.inPos )
      Coil( "Unit1.Em5.ControlNodes".transferPnPRight."step".action1[160] )
   END_RUNG
   RUNG wire#w1
      Contact( "Unit1.Em5.ControlNodes".cm.softcam.transferPnPRightAxisY.pos00_wait.inPos )
      Coil( "Unit1.Em5.ControlNodes".transferPnPRight."step".transition1[160] )
   END_RUNG
   RUNG wire#w1
      Contact( "Unit1.Em5.ControlNodes".transferPnPRight."step".transition1[160] )
      { S7_Templates := "time_type := Time" } #statTonTime[160].TON(pt := #delayTime, et =>)
      Move(in := #JOB_1_STEP_70, out1 => "Unit1.Em5.ControlNodes".transferPnPRight.sequence.status.nextStep)
   END_RUNG
   // the same network as SCL:
   #_w1 := ("Unit1.Em5.ControlNodes".transferPnPRight.sequence.status.currentStep = #JOB_1_STEP_60) AND "Unit1.Em5.ControlNodes".transferPnPRight.sequence.status.seqActive;
   "Unit1.Em5.ControlNodes".transferPnPRight."step".action1[160] := #_w1 AND NOT "Unit1.Em5.ControlNodes".cm.softcam.transferPnPRightAxisY.pos00_wait.inPos;
   "Unit1.Em5.ControlNodes".transferPnPRight."step".transition1[160] := #_w1 AND "Unit1.Em5.ControlNodes".cm.softcam.transferPnPRightAxisY.pos00_wait.inPos;
   #statTonTime[160].TON(IN := #_w1 AND "Unit1.Em5.ControlNodes".transferPnPRight."step".transition1[160],
                         PT := #delayTime);
   IF #statTonTime[160].Q THEN
       "Unit1.Em5.ControlNodes".transferPnPRight.sequence.status.nextStep := #JOB_1_STEP_70;
   END_IF;
END_REGION

REGION Network 11: Step[170] : Transfer PP Right Z-Axis Wait Position
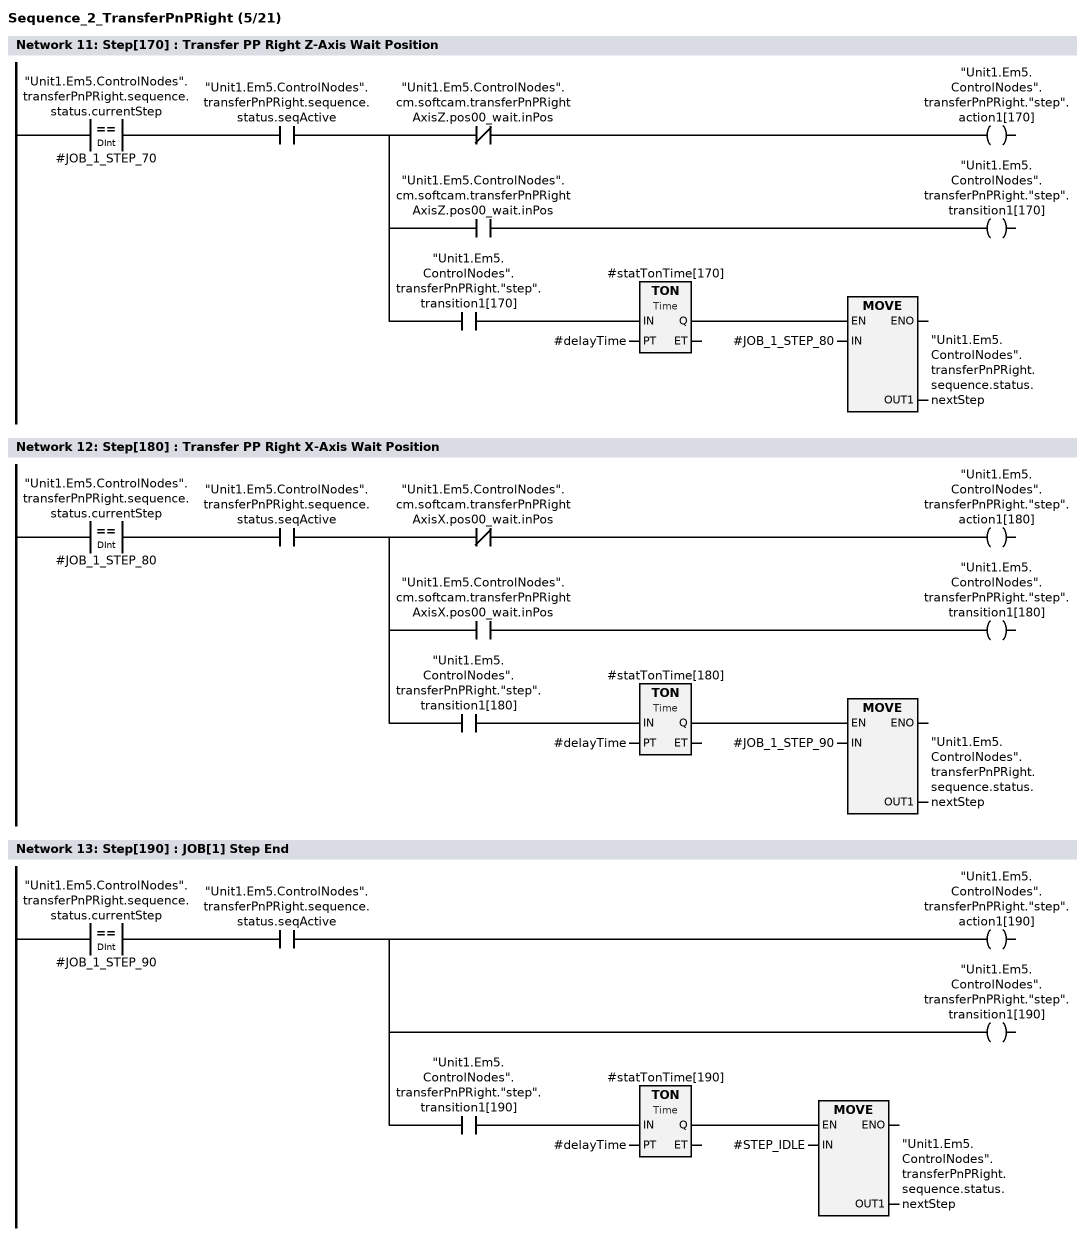
   RUNG wire#powerrail
      { S7_Templates := "SrcType := DInt" } EQ_Contact(in1 := "Unit1.Em5.ControlNodes".transferPnPRight.sequence.status.currentStep, in2 := #JOB_1_STEP_70)
      Contact( "Unit1.Em5.ControlNodes".transferPnPRight.sequence.status.seqActive )
      wire#w1
      I_Contact( "Unit1.Em5.ControlNodes".cm.softcam.transferPnPRightAxisZ.pos00_wait.inPos )
      Coil( "Unit1.Em5.ControlNodes".transferPnPRight."step".action1[170] )
   END_RUNG
   RUNG wire#w1
      Contact( "Unit1.Em5.ControlNodes".cm.softcam.transferPnPRightAxisZ.pos00_wait.inPos )
      Coil( "Unit1.Em5.ControlNodes".transferPnPRight."step".transition1[170] )
   END_RUNG
   RUNG wire#w1
      Contact( "Unit1.Em5.ControlNodes".transferPnPRight."step".transition1[170] )
      { S7_Templates := "time_type := Time" } #statTonTime[170].TON(pt := #delayTime, et =>)
      Move(in := #JOB_1_STEP_80, out1 => "Unit1.Em5.ControlNodes".transferPnPRight.sequence.status.nextStep)
   END_RUNG
   // the same network as SCL:
   #_w1 := ("Unit1.Em5.ControlNodes".transferPnPRight.sequence.status.currentStep = #JOB_1_STEP_70) AND "Unit1.Em5.ControlNodes".transferPnPRight.sequence.status.seqActive;
   "Unit1.Em5.ControlNodes".transferPnPRight."step".action1[170] := #_w1 AND NOT "Unit1.Em5.ControlNodes".cm.softcam.transferPnPRightAxisZ.pos00_wait.inPos;
   "Unit1.Em5.ControlNodes".transferPnPRight."step".transition1[170] := #_w1 AND "Unit1.Em5.ControlNodes".cm.softcam.transferPnPRightAxisZ.pos00_wait.inPos;
   #statTonTime[170].TON(IN := #_w1 AND "Unit1.Em5.ControlNodes".transferPnPRight."step".transition1[170],
                         PT := #delayTime);
   IF #statTonTime[170].Q THEN
       "Unit1.Em5.ControlNodes".transferPnPRight.sequence.status.nextStep := #JOB_1_STEP_80;
   END_IF;
END_REGION

REGION Network 12: Step[180] : Transfer PP Right X-Axis Wait Position
   RUNG wire#powerrail
      { S7_Templates := "SrcType := DInt" } EQ_Contact(in1 := "Unit1.Em5.ControlNodes".transferPnPRight.sequence.status.currentStep, in2 := #JOB_1_STEP_80)
      Contact( "Unit1.Em5.ControlNodes".transferPnPRight.sequence.status.seqActive )
      wire#w1
      I_Contact( "Unit1.Em5.ControlNodes".cm.softcam.transferPnPRightAxisX.pos00_wait.inPos )
      Coil( "Unit1.Em5.ControlNodes".transferPnPRight."step".action1[180] )
   END_RUNG
   RUNG wire#w1
      Contact( "Unit1.Em5.ControlNodes".cm.softcam.transferPnPRightAxisX.pos00_wait.inPos )
      Coil( "Unit1.Em5.ControlNodes".transferPnPRight."step".transition1[180] )
   END_RUNG
   RUNG wire#w1
      Contact( "Unit1.Em5.ControlNodes".transferPnPRight."step".transition1[180] )
      { S7_Templates := "time_type := Time" } #statTonTime[180].TON(pt := #delayTime, et =>)
      Move(in := #JOB_1_STEP_90, out1 => "Unit1.Em5.ControlNodes".transferPnPRight.sequence.status.nextStep)
   END_RUNG
   // the same network as SCL:
   #_w1 := ("Unit1.Em5.ControlNodes".transferPnPRight.sequence.status.currentStep = #JOB_1_STEP_80) AND "Unit1.Em5.ControlNodes".transferPnPRight.sequence.status.seqActive;
   "Unit1.Em5.ControlNodes".transferPnPRight."step".action1[180] := #_w1 AND NOT "Unit1.Em5.ControlNodes".cm.softcam.transferPnPRightAxisX.pos00_wait.inPos;
   "Unit1.Em5.ControlNodes".transferPnPRight."step".transition1[180] := #_w1 AND "Unit1.Em5.ControlNodes".cm.softcam.transferPnPRightAxisX.pos00_wait.inPos;
   #statTonTime[180].TON(IN := #_w1 AND "Unit1.Em5.ControlNodes".transferPnPRight."step".transition1[180],
                         PT := #delayTime);
   IF #statTonTime[180].Q THEN
       "Unit1.Em5.ControlNodes".transferPnPRight.sequence.status.nextStep := #JOB_1_STEP_90;
   END_IF;
END_REGION

REGION Network 13: Step[190] : JOB[1] Step End
   RUNG wire#powerrail
      { S7_Templates := "SrcType := DInt" } EQ_Contact(in1 := "Unit1.Em5.ControlNodes".transferPnPRight.sequence.status.currentStep, in2 := #JOB_1_STEP_90)
      Contact( "Unit1.Em5.ControlNodes".transferPnPRight.sequence.status.seqActive )
      wire#w1
      Coil( "Unit1.Em5.ControlNodes".transferPnPRight."step".action1[190] )
   END_RUNG
   RUNG wire#w1
      Coil( "Unit1.Em5.ControlNodes".transferPnPRight."step".transition1[190] )
   END_RUNG
   RUNG wire#w1
      Contact( "Unit1.Em5.ControlNodes".transferPnPRight."step".transition1[190] )
      { S7_Templates := "time_type := Time" } #statTonTime[190].TON(pt := #delayTime, et =>)
      Move(in := #STEP_IDLE, out1 => "Unit1.Em5.ControlNodes".transferPnPRight.sequence.status.nextStep)
   END_RUNG
   // the same network as SCL:
   "Unit1.Em5.ControlNodes".transferPnPRight."step".action1[190] := ("Unit1.Em5.ControlNodes".transferPnPRight.sequence.status.currentStep = #JOB_1_STEP_90) AND "Unit1.Em5.ControlNodes".transferPnPRight.sequence.status.seqActive;
   "Unit1.Em5.ControlNodes".transferPnPRight."step".transition1[190] := ("Unit1.Em5.ControlNodes".transferPnPRight.sequence.status.currentStep = #JOB_1_STEP_90) AND "Unit1.Em5.ControlNodes".transferPnPRight.sequence.status.seqActive;
   #statTonTime[190].TON(IN := ("Unit1.Em5.ControlNodes".transferPnPRight.sequence.status.currentStep = #JOB_1_STEP_90) AND "Unit1.Em5.ControlNodes".transferPnPRight.sequence.status.seqActive AND "Unit1.Em5.ControlNodes".transferPnPRight."step".transition1[190],
                         PT := #delayTime);
   IF #statTonTime[190].Q THEN
       "Unit1.Em5.ControlNodes".transferPnPRight.sequence.status.nextStep := #STEP_IDLE;
   END_IF;
END_REGION

REGION Network 14: *********** JOB[2] HIPOT & THICKNESS JR GET=AUTO-[A] ************
END_REGION

REGION Network 15: Step[201] : JOB[2] Condition
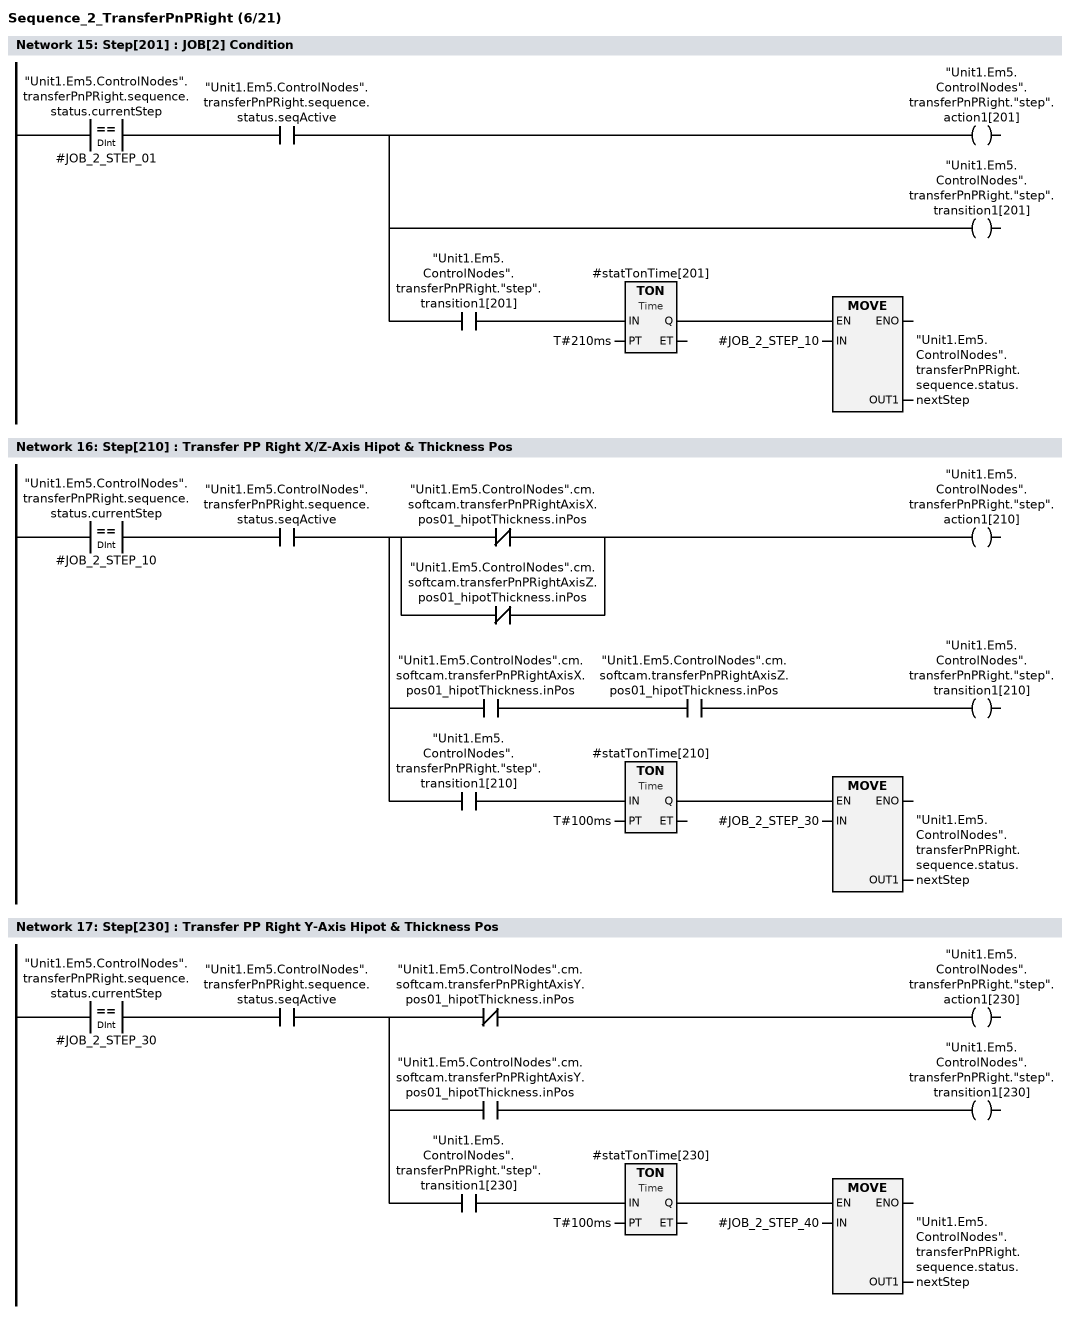
   RUNG wire#powerrail
      { S7_Templates := "SrcType := DInt" } EQ_Contact(in1 := "Unit1.Em5.ControlNodes".transferPnPRight.sequence.status.currentStep, in2 := #JOB_2_STEP_01)
      Contact( "Unit1.Em5.ControlNodes".transferPnPRight.sequence.status.seqActive )
      wire#w1
      Coil( "Unit1.Em5.ControlNodes".transferPnPRight."step".action1[201] )
   END_RUNG
   RUNG wire#w1
      Coil( "Unit1.Em5.ControlNodes".transferPnPRight."step".transition1[201] )
   END_RUNG
   RUNG wire#w1
      Contact( "Unit1.Em5.ControlNodes".transferPnPRight."step".transition1[201] )
      { S7_Templates := "time_type := Time" } #statTonTime[201].TON(pt := T#210ms, et =>)
      Move(in := #JOB_2_STEP_10, out1 => "Unit1.Em5.ControlNodes".transferPnPRight.sequence.status.nextStep)
   END_RUNG
   // the same network as SCL:
   "Unit1.Em5.ControlNodes".transferPnPRight."step".action1[201] := ("Unit1.Em5.ControlNodes".transferPnPRight.sequence.status.currentStep = #JOB_2_STEP_01) AND "Unit1.Em5.ControlNodes".transferPnPRight.sequence.status.seqActive;
   "Unit1.Em5.ControlNodes".transferPnPRight."step".transition1[201] := ("Unit1.Em5.ControlNodes".transferPnPRight.sequence.status.currentStep = #JOB_2_STEP_01) AND "Unit1.Em5.ControlNodes".transferPnPRight.sequence.status.seqActive;
   #statTonTime[201].TON(IN := ("Unit1.Em5.ControlNodes".transferPnPRight.sequence.status.currentStep = #JOB_2_STEP_01) AND "Unit1.Em5.ControlNodes".transferPnPRight.sequence.status.seqActive AND "Unit1.Em5.ControlNodes".transferPnPRight."step".transition1[201],
                         PT := T#210ms);
   IF #statTonTime[201].Q THEN
       "Unit1.Em5.ControlNodes".transferPnPRight.sequence.status.nextStep := #JOB_2_STEP_10;
   END_IF;
END_REGION

REGION Network 16: Step[210] : Transfer PP Right X/Z-Axis Hipot & Thickness Pos
   RUNG wire#powerrail
      { S7_Templates := "SrcType := DInt" } EQ_Contact(in1 := "Unit1.Em5.ControlNodes".transferPnPRight.sequence.status.currentStep, in2 := #JOB_2_STEP_10)
      Contact( "Unit1.Em5.ControlNodes".transferPnPRight.sequence.status.seqActive )
      wire#w1
      I_Contact( "Unit1.Em5.ControlNodes".cm.softcam.transferPnPRightAxisX.pos01_hipotThickness.inPos )
      wire#w2
      Coil( "Unit1.Em5.ControlNodes".transferPnPRight."step".action1[210] )
   END_RUNG
   RUNG wire#w1
      I_Contact( "Unit1.Em5.ControlNodes".cm.softcam.transferPnPRightAxisZ.pos01_hipotThickness.inPos )
   END_RUNG wire#w2
   RUNG wire#w1
      Contact( "Unit1.Em5.ControlNodes".cm.softcam.transferPnPRightAxisX.pos01_hipotThickness.inPos )
      Contact( "Unit1.Em5.ControlNodes".cm.softcam.transferPnPRightAxisZ.pos01_hipotThickness.inPos )
      Coil( "Unit1.Em5.ControlNodes".transferPnPRight."step".transition1[210] )
   END_RUNG
   RUNG wire#w1
      Contact( "Unit1.Em5.ControlNodes".transferPnPRight."step".transition1[210] )
      { S7_Templates := "time_type := Time" } #statTonTime[210].TON(pt := T#100ms, et =>)
      Move(in := #JOB_2_STEP_30, out1 => "Unit1.Em5.ControlNodes".transferPnPRight.sequence.status.nextStep)
   END_RUNG
   // the same network as SCL:
   #_w1 := ("Unit1.Em5.ControlNodes".transferPnPRight.sequence.status.currentStep = #JOB_2_STEP_10) AND "Unit1.Em5.ControlNodes".transferPnPRight.sequence.status.seqActive;
   "Unit1.Em5.ControlNodes".transferPnPRight."step".action1[210] := #_w1 AND (NOT "Unit1.Em5.ControlNodes".cm.softcam.transferPnPRightAxisX.pos01_hipotThickness.inPos OR NOT "Unit1.Em5.ControlNodes".cm.softcam.transferPnPRightAxisZ.pos01_hipotThickness.inPos);
   "Unit1.Em5.ControlNodes".transferPnPRight."step".transition1[210] := #_w1 AND "Unit1.Em5.ControlNodes".cm.softcam.transferPnPRightAxisX.pos01_hipotThickness.inPos AND "Unit1.Em5.ControlNodes".cm.softcam.transferPnPRightAxisZ.pos01_hipotThickness.inPos;
   #statTonTime[210].TON(IN := #_w1 AND "Unit1.Em5.ControlNodes".transferPnPRight."step".transition1[210],
                         PT := T#100ms);
   IF #statTonTime[210].Q THEN
       "Unit1.Em5.ControlNodes".transferPnPRight.sequence.status.nextStep := #JOB_2_STEP_30;
   END_IF;
END_REGION

REGION Network 17: Step[230] : Transfer PP Right Y-Axis Hipot & Thickness Pos
   RUNG wire#powerrail
      { S7_Templates := "SrcType := DInt" } EQ_Contact(in1 := "Unit1.Em5.ControlNodes".transferPnPRight.sequence.status.currentStep, in2 := #JOB_2_STEP_30)
      Contact( "Unit1.Em5.ControlNodes".transferPnPRight.sequence.status.seqActive )
      wire#w1
      I_Contact( "Unit1.Em5.ControlNodes".cm.softcam.transferPnPRightAxisY.pos01_hipotThickness.inPos )
      Coil( "Unit1.Em5.ControlNodes".transferPnPRight."step".action1[230] )
   END_RUNG
   RUNG wire#w1
      Contact( "Unit1.Em5.ControlNodes".cm.softcam.transferPnPRightAxisY.pos01_hipotThickness.inPos )
      Coil( "Unit1.Em5.ControlNodes".transferPnPRight."step".transition1[230] )
   END_RUNG
   RUNG wire#w1
      Contact( "Unit1.Em5.ControlNodes".transferPnPRight."step".transition1[230] )
      { S7_Templates := "time_type := Time" } #statTonTime[230].TON(pt := T#100ms, et =>)
      Move(in := #JOB_2_STEP_40, out1 => "Unit1.Em5.ControlNodes".transferPnPRight.sequence.status.nextStep)
   END_RUNG
   // the same network as SCL:
   #_w1 := ("Unit1.Em5.ControlNodes".transferPnPRight.sequence.status.currentStep = #JOB_2_STEP_30) AND "Unit1.Em5.ControlNodes".transferPnPRight.sequence.status.seqActive;
   "Unit1.Em5.ControlNodes".transferPnPRight."step".action1[230] := #_w1 AND NOT "Unit1.Em5.ControlNodes".cm.softcam.transferPnPRightAxisY.pos01_hipotThickness.inPos;
   "Unit1.Em5.ControlNodes".transferPnPRight."step".transition1[230] := #_w1 AND "Unit1.Em5.ControlNodes".cm.softcam.transferPnPRightAxisY.pos01_hipotThickness.inPos;
   #statTonTime[230].TON(IN := #_w1 AND "Unit1.Em5.ControlNodes".transferPnPRight."step".transition1[230],
                         PT := T#100ms);
   IF #statTonTime[230].Q THEN
       "Unit1.Em5.ControlNodes".transferPnPRight.sequence.status.nextStep := #JOB_2_STEP_40;
   END_IF;
END_REGION

REGION Network 18: Step[240] : Transfer PP Right Clamp Close
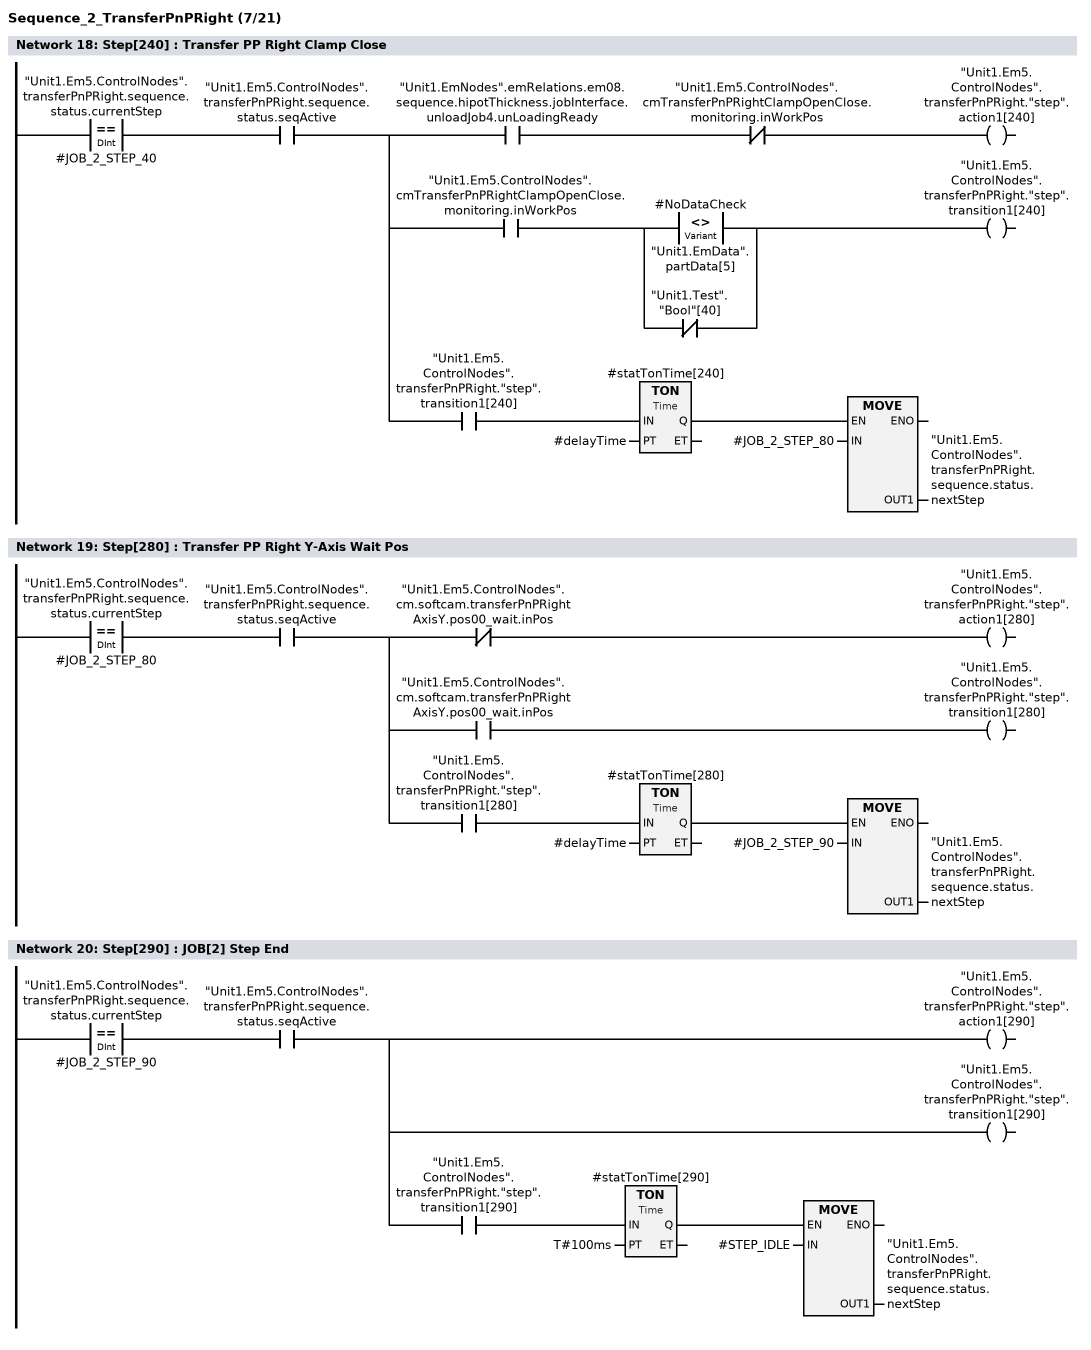
   RUNG wire#powerrail
      { S7_Templates := "SrcType := DInt" } EQ_Contact(in1 := "Unit1.Em5.ControlNodes".transferPnPRight.sequence.status.currentStep, in2 := #JOB_2_STEP_40)
      Contact( "Unit1.Em5.ControlNodes".transferPnPRight.sequence.status.seqActive )
      wire#w1
      Contact( "Unit1.EmNodes".emRelations.em08.sequence.hipotThickness.jobInterface.unloadJob4.unLoadingReady )
      I_Contact( "Unit1.Em5.ControlNodes".cmTransferPnPRightClampOpenClose.monitoring.inWorkPos )
      Coil( "Unit1.Em5.ControlNodes".transferPnPRight."step".action1[240] )
   END_RUNG
   RUNG wire#w1
      Contact( "Unit1.Em5.ControlNodes".cmTransferPnPRightClampOpenClose.monitoring.inWorkPos )
      wire#w2
      { S7_Templates := "SrcType := Variant" } NE_Contact(in1 := #NoDataCheck, in2 := "Unit1.EmData".partData[5])
      wire#w3
      Coil( "Unit1.Em5.ControlNodes".transferPnPRight."step".transition1[240] )
   END_RUNG
   RUNG wire#w2
      I_Contact( "Unit1.Test"."Bool"[40] )
   END_RUNG wire#w3
   RUNG wire#w1
      Contact( "Unit1.Em5.ControlNodes".transferPnPRight."step".transition1[240] )
      { S7_Templates := "time_type := Time" } #statTonTime[240].TON(pt := #delayTime, et =>)
      Move(in := #JOB_2_STEP_80, out1 => "Unit1.Em5.ControlNodes".transferPnPRight.sequence.status.nextStep)
   END_RUNG
   // the same network as SCL:
   #_w1 := ("Unit1.Em5.ControlNodes".transferPnPRight.sequence.status.currentStep = #JOB_2_STEP_40) AND "Unit1.Em5.ControlNodes".transferPnPRight.sequence.status.seqActive;
   "Unit1.Em5.ControlNodes".transferPnPRight."step".action1[240] := #_w1 AND "Unit1.EmNodes".emRelations.em08.sequence.hipotThickness.jobInterface.unloadJob4.unLoadingReady AND NOT "Unit1.Em5.ControlNodes".cmTransferPnPRightClampOpenClose.monitoring.inWorkPos;
   "Unit1.Em5.ControlNodes".transferPnPRight."step".transition1[240] := #_w1 AND "Unit1.Em5.ControlNodes".cmTransferPnPRightClampOpenClose.monitoring.inWorkPos AND ((#NoDataCheck <> "Unit1.EmData".partData[5]) OR NOT "Unit1.Test"."Bool"[40]);
   #statTonTime[240].TON(IN := #_w1 AND "Unit1.Em5.ControlNodes".transferPnPRight."step".transition1[240],
                         PT := #delayTime);
   IF #statTonTime[240].Q THEN
       "Unit1.Em5.ControlNodes".transferPnPRight.sequence.status.nextStep := #JOB_2_STEP_80;
   END_IF;
END_REGION

REGION Network 19: Step[280] : Transfer PP Right Y-Axis Wait Pos
   RUNG wire#powerrail
      { S7_Templates := "SrcType := DInt" } EQ_Contact(in1 := "Unit1.Em5.ControlNodes".transferPnPRight.sequence.status.currentStep, in2 := #JOB_2_STEP_80)
      Contact( "Unit1.Em5.ControlNodes".transferPnPRight.sequence.status.seqActive )
      wire#w1
      I_Contact( "Unit1.Em5.ControlNodes".cm.softcam.transferPnPRightAxisY.pos00_wait.inPos )
      Coil( "Unit1.Em5.ControlNodes".transferPnPRight."step".action1[280] )
   END_RUNG
   RUNG wire#w1
      Contact( "Unit1.Em5.ControlNodes".cm.softcam.transferPnPRightAxisY.pos00_wait.inPos )
      Coil( "Unit1.Em5.ControlNodes".transferPnPRight."step".transition1[280] )
   END_RUNG
   RUNG wire#w1
      Contact( "Unit1.Em5.ControlNodes".transferPnPRight."step".transition1[280] )
      { S7_Templates := "time_type := Time" } #statTonTime[280].TON(pt := #delayTime, et =>)
      Move(in := #JOB_2_STEP_90, out1 => "Unit1.Em5.ControlNodes".transferPnPRight.sequence.status.nextStep)
   END_RUNG
   // the same network as SCL:
   #_w1 := ("Unit1.Em5.ControlNodes".transferPnPRight.sequence.status.currentStep = #JOB_2_STEP_80) AND "Unit1.Em5.ControlNodes".transferPnPRight.sequence.status.seqActive;
   "Unit1.Em5.ControlNodes".transferPnPRight."step".action1[280] := #_w1 AND NOT "Unit1.Em5.ControlNodes".cm.softcam.transferPnPRightAxisY.pos00_wait.inPos;
   "Unit1.Em5.ControlNodes".transferPnPRight."step".transition1[280] := #_w1 AND "Unit1.Em5.ControlNodes".cm.softcam.transferPnPRightAxisY.pos00_wait.inPos;
   #statTonTime[280].TON(IN := #_w1 AND "Unit1.Em5.ControlNodes".transferPnPRight."step".transition1[280],
                         PT := #delayTime);
   IF #statTonTime[280].Q THEN
       "Unit1.Em5.ControlNodes".transferPnPRight.sequence.status.nextStep := #JOB_2_STEP_90;
   END_IF;
END_REGION

REGION Network 20: Step[290] : JOB[2] Step End
   RUNG wire#powerrail
      { S7_Templates := "SrcType := DInt" } EQ_Contact(in1 := "Unit1.Em5.ControlNodes".transferPnPRight.sequence.status.currentStep, in2 := #JOB_2_STEP_90)
      Contact( "Unit1.Em5.ControlNodes".transferPnPRight.sequence.status.seqActive )
      wire#w1
      Coil( "Unit1.Em5.ControlNodes".transferPnPRight."step".action1[290] )
   END_RUNG
   RUNG wire#w1
      Coil( "Unit1.Em5.ControlNodes".transferPnPRight."step".transition1[290] )
   END_RUNG
   RUNG wire#w1
      Contact( "Unit1.Em5.ControlNodes".transferPnPRight."step".transition1[290] )
      { S7_Templates := "time_type := Time" } #statTonTime[290].TON(pt := T#100ms, et =>)
      Move(in := #STEP_IDLE, out1 => "Unit1.Em5.ControlNodes".transferPnPRight.sequence.status.nextStep)
   END_RUNG
   // the same network as SCL:
   "Unit1.Em5.ControlNodes".transferPnPRight."step".action1[290] := ("Unit1.Em5.ControlNodes".transferPnPRight.sequence.status.currentStep = #JOB_2_STEP_90) AND "Unit1.Em5.ControlNodes".transferPnPRight.sequence.status.seqActive;
   "Unit1.Em5.ControlNodes".transferPnPRight."step".transition1[290] := ("Unit1.Em5.ControlNodes".transferPnPRight.sequence.status.currentStep = #JOB_2_STEP_90) AND "Unit1.Em5.ControlNodes".transferPnPRight.sequence.status.seqActive;
   #statTonTime[290].TON(IN := ("Unit1.Em5.ControlNodes".transferPnPRight.sequence.status.currentStep = #JOB_2_STEP_90) AND "Unit1.Em5.ControlNodes".transferPnPRight.sequence.status.seqActive AND "Unit1.Em5.ControlNodes".transferPnPRight."step".transition1[290],
                         PT := T#100ms);
   IF #statTonTime[290].Q THEN
       "Unit1.Em5.ControlNodes".transferPnPRight.sequence.status.nextStep := #STEP_IDLE;
   END_IF;
END_REGION

REGION Network 21: **************** JOB[3] VISION JR PUT=AUTO-[A] *****************
END_REGION

REGION Network 22: Step[301] : JOB[3] Condition
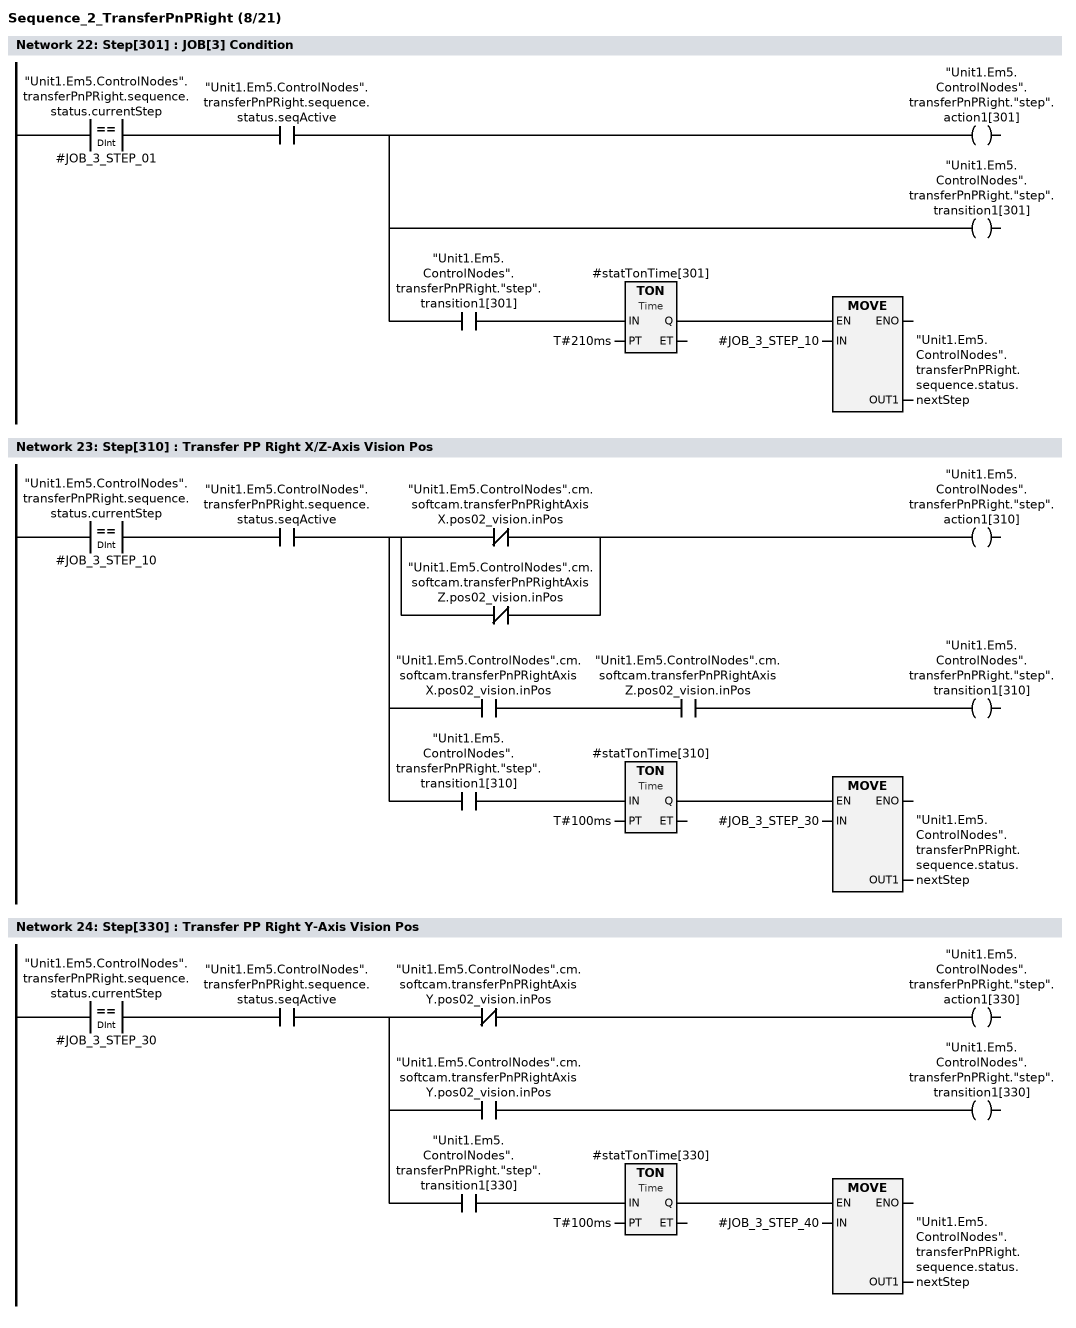
   RUNG wire#powerrail
      { S7_Templates := "SrcType := DInt" } EQ_Contact(in1 := "Unit1.Em5.ControlNodes".transferPnPRight.sequence.status.currentStep, in2 := #JOB_3_STEP_01)
      Contact( "Unit1.Em5.ControlNodes".transferPnPRight.sequence.status.seqActive )
      wire#w1
      Coil( "Unit1.Em5.ControlNodes".transferPnPRight."step".action1[301] )
   END_RUNG
   RUNG wire#w1
      Coil( "Unit1.Em5.ControlNodes".transferPnPRight."step".transition1[301] )
   END_RUNG
   RUNG wire#w1
      Contact( "Unit1.Em5.ControlNodes".transferPnPRight."step".transition1[301] )
      { S7_Templates := "time_type := Time" } #statTonTime[301].TON(pt := T#210ms, et =>)
      Move(in := #JOB_3_STEP_10, out1 => "Unit1.Em5.ControlNodes".transferPnPRight.sequence.status.nextStep)
   END_RUNG
   // the same network as SCL:
   "Unit1.Em5.ControlNodes".transferPnPRight."step".action1[301] := ("Unit1.Em5.ControlNodes".transferPnPRight.sequence.status.currentStep = #JOB_3_STEP_01) AND "Unit1.Em5.ControlNodes".transferPnPRight.sequence.status.seqActive;
   "Unit1.Em5.ControlNodes".transferPnPRight."step".transition1[301] := ("Unit1.Em5.ControlNodes".transferPnPRight.sequence.status.currentStep = #JOB_3_STEP_01) AND "Unit1.Em5.ControlNodes".transferPnPRight.sequence.status.seqActive;
   #statTonTime[301].TON(IN := ("Unit1.Em5.ControlNodes".transferPnPRight.sequence.status.currentStep = #JOB_3_STEP_01) AND "Unit1.Em5.ControlNodes".transferPnPRight.sequence.status.seqActive AND "Unit1.Em5.ControlNodes".transferPnPRight."step".transition1[301],
                         PT := T#210ms);
   IF #statTonTime[301].Q THEN
       "Unit1.Em5.ControlNodes".transferPnPRight.sequence.status.nextStep := #JOB_3_STEP_10;
   END_IF;
END_REGION

REGION Network 23: Step[310] : Transfer PP Right X/Z-Axis Vision Pos
   RUNG wire#powerrail
      { S7_Templates := "SrcType := DInt" } EQ_Contact(in1 := "Unit1.Em5.ControlNodes".transferPnPRight.sequence.status.currentStep, in2 := #JOB_3_STEP_10)
      Contact( "Unit1.Em5.ControlNodes".transferPnPRight.sequence.status.seqActive )
      wire#w1
      I_Contact( "Unit1.Em5.ControlNodes".cm.softcam.transferPnPRightAxisX.pos02_vision.inPos )
      wire#w2
      Coil( "Unit1.Em5.ControlNodes".transferPnPRight."step".action1[310] )
   END_RUNG
   RUNG wire#w1
      I_Contact( "Unit1.Em5.ControlNodes".cm.softcam.transferPnPRightAxisZ.pos02_vision.inPos )
   END_RUNG wire#w2
   RUNG wire#w1
      Contact( "Unit1.Em5.ControlNodes".cm.softcam.transferPnPRightAxisX.pos02_vision.inPos )
      Contact( "Unit1.Em5.ControlNodes".cm.softcam.transferPnPRightAxisZ.pos02_vision.inPos )
      Coil( "Unit1.Em5.ControlNodes".transferPnPRight."step".transition1[310] )
   END_RUNG
   RUNG wire#w1
      Contact( "Unit1.Em5.ControlNodes".transferPnPRight."step".transition1[310] )
      { S7_Templates := "time_type := Time" } #statTonTime[310].TON(pt := T#100ms, et =>)
      Move(in := #JOB_3_STEP_30, out1 => "Unit1.Em5.ControlNodes".transferPnPRight.sequence.status.nextStep)
   END_RUNG
   // the same network as SCL:
   #_w1 := ("Unit1.Em5.ControlNodes".transferPnPRight.sequence.status.currentStep = #JOB_3_STEP_10) AND "Unit1.Em5.ControlNodes".transferPnPRight.sequence.status.seqActive;
   "Unit1.Em5.ControlNodes".transferPnPRight."step".action1[310] := #_w1 AND (NOT "Unit1.Em5.ControlNodes".cm.softcam.transferPnPRightAxisX.pos02_vision.inPos OR NOT "Unit1.Em5.ControlNodes".cm.softcam.transferPnPRightAxisZ.pos02_vision.inPos);
   "Unit1.Em5.ControlNodes".transferPnPRight."step".transition1[310] := #_w1 AND "Unit1.Em5.ControlNodes".cm.softcam.transferPnPRightAxisX.pos02_vision.inPos AND "Unit1.Em5.ControlNodes".cm.softcam.transferPnPRightAxisZ.pos02_vision.inPos;
   #statTonTime[310].TON(IN := #_w1 AND "Unit1.Em5.ControlNodes".transferPnPRight."step".transition1[310],
                         PT := T#100ms);
   IF #statTonTime[310].Q THEN
       "Unit1.Em5.ControlNodes".transferPnPRight.sequence.status.nextStep := #JOB_3_STEP_30;
   END_IF;
END_REGION

REGION Network 24: Step[330] : Transfer PP Right Y-Axis Vision Pos
   RUNG wire#powerrail
      { S7_Templates := "SrcType := DInt" } EQ_Contact(in1 := "Unit1.Em5.ControlNodes".transferPnPRight.sequence.status.currentStep, in2 := #JOB_3_STEP_30)
      Contact( "Unit1.Em5.ControlNodes".transferPnPRight.sequence.status.seqActive )
      wire#w1
      I_Contact( "Unit1.Em5.ControlNodes".cm.softcam.transferPnPRightAxisY.pos02_vision.inPos )
      Coil( "Unit1.Em5.ControlNodes".transferPnPRight."step".action1[330] )
   END_RUNG
   RUNG wire#w1
      Contact( "Unit1.Em5.ControlNodes".cm.softcam.transferPnPRightAxisY.pos02_vision.inPos )
      Coil( "Unit1.Em5.ControlNodes".transferPnPRight."step".transition1[330] )
   END_RUNG
   RUNG wire#w1
      Contact( "Unit1.Em5.ControlNodes".transferPnPRight."step".transition1[330] )
      { S7_Templates := "time_type := Time" } #statTonTime[330].TON(pt := T#100ms, et =>)
      Move(in := #JOB_3_STEP_40, out1 => "Unit1.Em5.ControlNodes".transferPnPRight.sequence.status.nextStep)
   END_RUNG
   // the same network as SCL:
   #_w1 := ("Unit1.Em5.ControlNodes".transferPnPRight.sequence.status.currentStep = #JOB_3_STEP_30) AND "Unit1.Em5.ControlNodes".transferPnPRight.sequence.status.seqActive;
   "Unit1.Em5.ControlNodes".transferPnPRight."step".action1[330] := #_w1 AND NOT "Unit1.Em5.ControlNodes".cm.softcam.transferPnPRightAxisY.pos02_vision.inPos;
   "Unit1.Em5.ControlNodes".transferPnPRight."step".transition1[330] := #_w1 AND "Unit1.Em5.ControlNodes".cm.softcam.transferPnPRightAxisY.pos02_vision.inPos;
   #statTonTime[330].TON(IN := #_w1 AND "Unit1.Em5.ControlNodes".transferPnPRight."step".transition1[330],
                         PT := T#100ms);
   IF #statTonTime[330].Q THEN
       "Unit1.Em5.ControlNodes".transferPnPRight.sequence.status.nextStep := #JOB_3_STEP_40;
   END_IF;
END_REGION

REGION Network 25: Step[340] : Transfer PP Right [Lift Up Request] => Vision Check
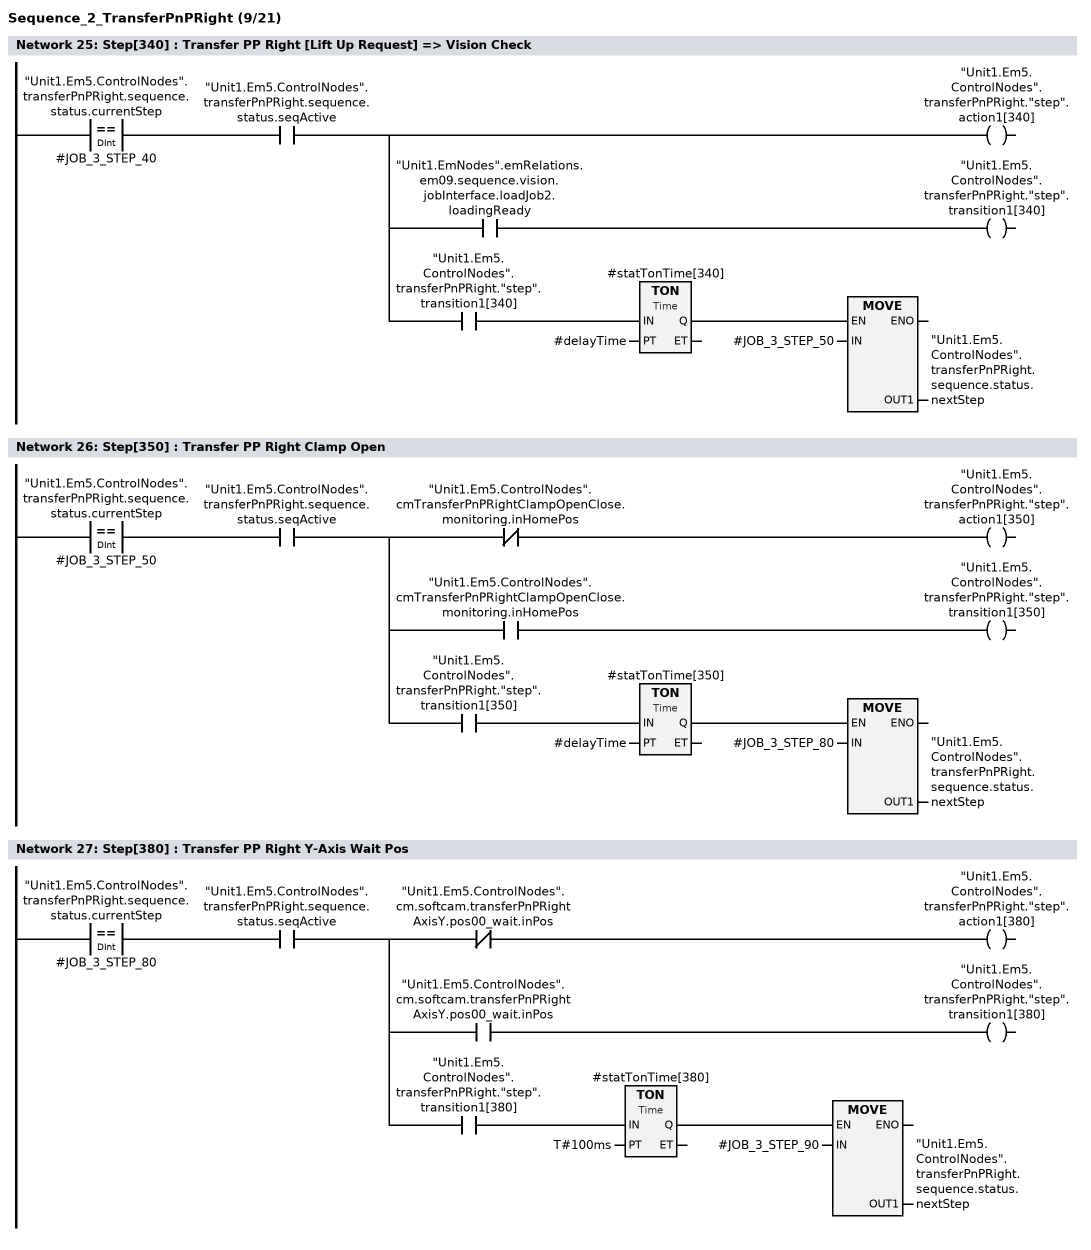
   RUNG wire#powerrail
      { S7_Templates := "SrcType := DInt" } EQ_Contact(in1 := "Unit1.Em5.ControlNodes".transferPnPRight.sequence.status.currentStep, in2 := #JOB_3_STEP_40)
      Contact( "Unit1.Em5.ControlNodes".transferPnPRight.sequence.status.seqActive )
      wire#w1
      Coil( "Unit1.Em5.ControlNodes".transferPnPRight."step".action1[340] )
   END_RUNG
   RUNG wire#w1
      Contact( "Unit1.EmNodes".emRelations.em09.sequence.vision.jobInterface.loadJob2.loadingReady )
      Coil( "Unit1.Em5.ControlNodes".transferPnPRight."step".transition1[340] )
   END_RUNG
   RUNG wire#w1
      Contact( "Unit1.Em5.ControlNodes".transferPnPRight."step".transition1[340] )
      { S7_Templates := "time_type := Time" } #statTonTime[340].TON(pt := #delayTime, et =>)
      Move(in := #JOB_3_STEP_50, out1 => "Unit1.Em5.ControlNodes".transferPnPRight.sequence.status.nextStep)
   END_RUNG
   // the same network as SCL:
   "Unit1.Em5.ControlNodes".transferPnPRight."step".action1[340] := ("Unit1.Em5.ControlNodes".transferPnPRight.sequence.status.currentStep = #JOB_3_STEP_40) AND "Unit1.Em5.ControlNodes".transferPnPRight.sequence.status.seqActive;
   "Unit1.Em5.ControlNodes".transferPnPRight."step".transition1[340] := ("Unit1.Em5.ControlNodes".transferPnPRight.sequence.status.currentStep = #JOB_3_STEP_40) AND "Unit1.Em5.ControlNodes".transferPnPRight.sequence.status.seqActive AND "Unit1.EmNodes".emRelations.em09.sequence.vision.jobInterface.loadJob2.loadingReady;
   #statTonTime[340].TON(IN := ("Unit1.Em5.ControlNodes".transferPnPRight.sequence.status.currentStep = #JOB_3_STEP_40) AND "Unit1.Em5.ControlNodes".transferPnPRight.sequence.status.seqActive AND "Unit1.Em5.ControlNodes".transferPnPRight."step".transition1[340],
                         PT := #delayTime);
   IF #statTonTime[340].Q THEN
       "Unit1.Em5.ControlNodes".transferPnPRight.sequence.status.nextStep := #JOB_3_STEP_50;
   END_IF;
END_REGION

REGION Network 26: Step[350] : Transfer PP Right Clamp Open
   RUNG wire#powerrail
      { S7_Templates := "SrcType := DInt" } EQ_Contact(in1 := "Unit1.Em5.ControlNodes".transferPnPRight.sequence.status.currentStep, in2 := #JOB_3_STEP_50)
      Contact( "Unit1.Em5.ControlNodes".transferPnPRight.sequence.status.seqActive )
      wire#w1
      I_Contact( "Unit1.Em5.ControlNodes".cmTransferPnPRightClampOpenClose.monitoring.inHomePos )
      Coil( "Unit1.Em5.ControlNodes".transferPnPRight."step".action1[350] )
   END_RUNG
   RUNG wire#w1
      Contact( "Unit1.Em5.ControlNodes".cmTransferPnPRightClampOpenClose.monitoring.inHomePos )
      Coil( "Unit1.Em5.ControlNodes".transferPnPRight."step".transition1[350] )
   END_RUNG
   RUNG wire#w1
      Contact( "Unit1.Em5.ControlNodes".transferPnPRight."step".transition1[350] )
      { S7_Templates := "time_type := Time" } #statTonTime[350].TON(pt := #delayTime, et =>)
      Move(in := #JOB_3_STEP_80, out1 => "Unit1.Em5.ControlNodes".transferPnPRight.sequence.status.nextStep)
   END_RUNG
   // the same network as SCL:
   #_w1 := ("Unit1.Em5.ControlNodes".transferPnPRight.sequence.status.currentStep = #JOB_3_STEP_50) AND "Unit1.Em5.ControlNodes".transferPnPRight.sequence.status.seqActive;
   "Unit1.Em5.ControlNodes".transferPnPRight."step".action1[350] := #_w1 AND NOT "Unit1.Em5.ControlNodes".cmTransferPnPRightClampOpenClose.monitoring.inHomePos;
   "Unit1.Em5.ControlNodes".transferPnPRight."step".transition1[350] := #_w1 AND "Unit1.Em5.ControlNodes".cmTransferPnPRightClampOpenClose.monitoring.inHomePos;
   #statTonTime[350].TON(IN := #_w1 AND "Unit1.Em5.ControlNodes".transferPnPRight."step".transition1[350],
                         PT := #delayTime);
   IF #statTonTime[350].Q THEN
       "Unit1.Em5.ControlNodes".transferPnPRight.sequence.status.nextStep := #JOB_3_STEP_80;
   END_IF;
END_REGION

REGION Network 27: Step[380] : Transfer PP Right Y-Axis Wait Pos
   RUNG wire#powerrail
      { S7_Templates := "SrcType := DInt" } EQ_Contact(in1 := "Unit1.Em5.ControlNodes".transferPnPRight.sequence.status.currentStep, in2 := #JOB_3_STEP_80)
      Contact( "Unit1.Em5.ControlNodes".transferPnPRight.sequence.status.seqActive )
      wire#w1
      I_Contact( "Unit1.Em5.ControlNodes".cm.softcam.transferPnPRightAxisY.pos00_wait.inPos )
      Coil( "Unit1.Em5.ControlNodes".transferPnPRight."step".action1[380] )
   END_RUNG
   RUNG wire#w1
      Contact( "Unit1.Em5.ControlNodes".cm.softcam.transferPnPRightAxisY.pos00_wait.inPos )
      Coil( "Unit1.Em5.ControlNodes".transferPnPRight."step".transition1[380] )
   END_RUNG
   RUNG wire#w1
      Contact( "Unit1.Em5.ControlNodes".transferPnPRight."step".transition1[380] )
      { S7_Templates := "time_type := Time" } #statTonTime[380].TON(pt := T#100ms, et =>)
      Move(in := #JOB_3_STEP_90, out1 => "Unit1.Em5.ControlNodes".transferPnPRight.sequence.status.nextStep)
   END_RUNG
   // the same network as SCL:
   #_w1 := ("Unit1.Em5.ControlNodes".transferPnPRight.sequence.status.currentStep = #JOB_3_STEP_80) AND "Unit1.Em5.ControlNodes".transferPnPRight.sequence.status.seqActive;
   "Unit1.Em5.ControlNodes".transferPnPRight."step".action1[380] := #_w1 AND NOT "Unit1.Em5.ControlNodes".cm.softcam.transferPnPRightAxisY.pos00_wait.inPos;
   "Unit1.Em5.ControlNodes".transferPnPRight."step".transition1[380] := #_w1 AND "Unit1.Em5.ControlNodes".cm.softcam.transferPnPRightAxisY.pos00_wait.inPos;
   #statTonTime[380].TON(IN := #_w1 AND "Unit1.Em5.ControlNodes".transferPnPRight."step".transition1[380],
                         PT := T#100ms);
   IF #statTonTime[380].Q THEN
       "Unit1.Em5.ControlNodes".transferPnPRight.sequence.status.nextStep := #JOB_3_STEP_90;
   END_IF;
END_REGION

REGION Network 28: Step[390] : JOB[3] Step End
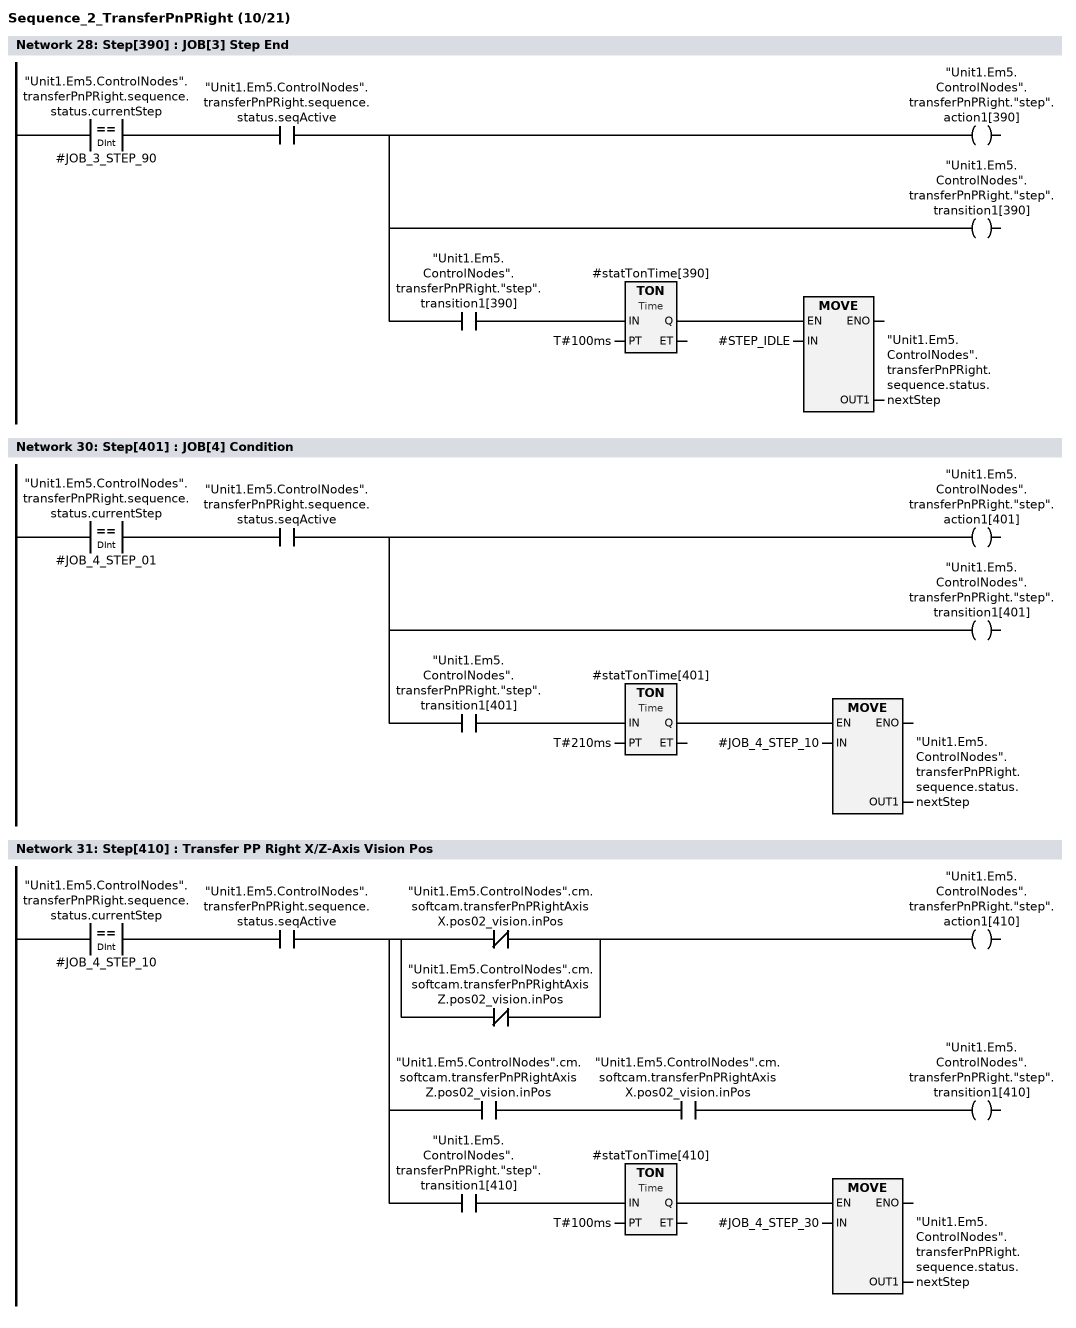
   RUNG wire#powerrail
      { S7_Templates := "SrcType := DInt" } EQ_Contact(in1 := "Unit1.Em5.ControlNodes".transferPnPRight.sequence.status.currentStep, in2 := #JOB_3_STEP_90)
      Contact( "Unit1.Em5.ControlNodes".transferPnPRight.sequence.status.seqActive )
      wire#w1
      Coil( "Unit1.Em5.ControlNodes".transferPnPRight."step".action1[390] )
   END_RUNG
   RUNG wire#w1
      Coil( "Unit1.Em5.ControlNodes".transferPnPRight."step".transition1[390] )
   END_RUNG
   RUNG wire#w1
      Contact( "Unit1.Em5.ControlNodes".transferPnPRight."step".transition1[390] )
      { S7_Templates := "time_type := Time" } #statTonTime[390].TON(pt := T#100ms, et =>)
      Move(in := #STEP_IDLE, out1 => "Unit1.Em5.ControlNodes".transferPnPRight.sequence.status.nextStep)
   END_RUNG
   // the same network as SCL:
   "Unit1.Em5.ControlNodes".transferPnPRight."step".action1[390] := ("Unit1.Em5.ControlNodes".transferPnPRight.sequence.status.currentStep = #JOB_3_STEP_90) AND "Unit1.Em5.ControlNodes".transferPnPRight.sequence.status.seqActive;
   "Unit1.Em5.ControlNodes".transferPnPRight."step".transition1[390] := ("Unit1.Em5.ControlNodes".transferPnPRight.sequence.status.currentStep = #JOB_3_STEP_90) AND "Unit1.Em5.ControlNodes".transferPnPRight.sequence.status.seqActive;
   #statTonTime[390].TON(IN := ("Unit1.Em5.ControlNodes".transferPnPRight.sequence.status.currentStep = #JOB_3_STEP_90) AND "Unit1.Em5.ControlNodes".transferPnPRight.sequence.status.seqActive AND "Unit1.Em5.ControlNodes".transferPnPRight."step".transition1[390],
                         PT := T#100ms);
   IF #statTonTime[390].Q THEN
       "Unit1.Em5.ControlNodes".transferPnPRight.sequence.status.nextStep := #STEP_IDLE;
   END_IF;
END_REGION

REGION Network 29: **************** JOB[4] VISION JR GET=AUTO-[A] *****************
END_REGION

REGION Network 30: Step[401] : JOB[4] Condition
   RUNG wire#powerrail
      { S7_Templates := "SrcType := DInt" } EQ_Contact(in1 := "Unit1.Em5.ControlNodes".transferPnPRight.sequence.status.currentStep, in2 := #JOB_4_STEP_01)
      Contact( "Unit1.Em5.ControlNodes".transferPnPRight.sequence.status.seqActive )
      wire#w1
      Coil( "Unit1.Em5.ControlNodes".transferPnPRight."step".action1[401] )
   END_RUNG
   RUNG wire#w1
      Coil( "Unit1.Em5.ControlNodes".transferPnPRight."step".transition1[401] )
   END_RUNG
   RUNG wire#w1
      Contact( "Unit1.Em5.ControlNodes".transferPnPRight."step".transition1[401] )
      { S7_Templates := "time_type := Time" } #statTonTime[401].TON(pt := T#210ms, et =>)
      Move(in := #JOB_4_STEP_10, out1 => "Unit1.Em5.ControlNodes".transferPnPRight.sequence.status.nextStep)
   END_RUNG
   // the same network as SCL:
   "Unit1.Em5.ControlNodes".transferPnPRight."step".action1[401] := ("Unit1.Em5.ControlNodes".transferPnPRight.sequence.status.currentStep = #JOB_4_STEP_01) AND "Unit1.Em5.ControlNodes".transferPnPRight.sequence.status.seqActive;
   "Unit1.Em5.ControlNodes".transferPnPRight."step".transition1[401] := ("Unit1.Em5.ControlNodes".transferPnPRight.sequence.status.currentStep = #JOB_4_STEP_01) AND "Unit1.Em5.ControlNodes".transferPnPRight.sequence.status.seqActive;
   #statTonTime[401].TON(IN := ("Unit1.Em5.ControlNodes".transferPnPRight.sequence.status.currentStep = #JOB_4_STEP_01) AND "Unit1.Em5.ControlNodes".transferPnPRight.sequence.status.seqActive AND "Unit1.Em5.ControlNodes".transferPnPRight."step".transition1[401],
                         PT := T#210ms);
   IF #statTonTime[401].Q THEN
       "Unit1.Em5.ControlNodes".transferPnPRight.sequence.status.nextStep := #JOB_4_STEP_10;
   END_IF;
END_REGION

REGION Network 31: Step[410] : Transfer PP Right X/Z-Axis Vision Pos
   RUNG wire#powerrail
      { S7_Templates := "SrcType := DInt" } EQ_Contact(in1 := "Unit1.Em5.ControlNodes".transferPnPRight.sequence.status.currentStep, in2 := #JOB_4_STEP_10)
      Contact( "Unit1.Em5.ControlNodes".transferPnPRight.sequence.status.seqActive )
      wire#w1
      I_Contact( "Unit1.Em5.ControlNodes".cm.softcam.transferPnPRightAxisX.pos02_vision.inPos )
      wire#w2
      Coil( "Unit1.Em5.ControlNodes".transferPnPRight."step".action1[410] )
   END_RUNG
   RUNG wire#w1
      I_Contact( "Unit1.Em5.ControlNodes".cm.softcam.transferPnPRightAxisZ.pos02_vision.inPos )
   END_RUNG wire#w2
   RUNG wire#w1
      Contact( "Unit1.Em5.ControlNodes".cm.softcam.transferPnPRightAxisZ.pos02_vision.inPos )
      Contact( "Unit1.Em5.ControlNodes".cm.softcam.transferPnPRightAxisX.pos02_vision.inPos )
      Coil( "Unit1.Em5.ControlNodes".transferPnPRight."step".transition1[410] )
   END_RUNG
   RUNG wire#w1
      Contact( "Unit1.Em5.ControlNodes".transferPnPRight."step".transition1[410] )
      { S7_Templates := "time_type := Time" } #statTonTime[410].TON(pt := T#100ms, et =>)
      Move(in := #JOB_4_STEP_30, out1 => "Unit1.Em5.ControlNodes".transferPnPRight.sequence.status.nextStep)
   END_RUNG
   // the same network as SCL:
   #_w1 := ("Unit1.Em5.ControlNodes".transferPnPRight.sequence.status.currentStep = #JOB_4_STEP_10) AND "Unit1.Em5.ControlNodes".transferPnPRight.sequence.status.seqActive;
   "Unit1.Em5.ControlNodes".transferPnPRight."step".action1[410] := #_w1 AND (NOT "Unit1.Em5.ControlNodes".cm.softcam.transferPnPRightAxisX.pos02_vision.inPos OR NOT "Unit1.Em5.ControlNodes".cm.softcam.transferPnPRightAxisZ.pos02_vision.inPos);
   "Unit1.Em5.ControlNodes".transferPnPRight."step".transition1[410] := #_w1 AND "Unit1.Em5.ControlNodes".cm.softcam.transferPnPRightAxisZ.pos02_vision.inPos AND "Unit1.Em5.ControlNodes".cm.softcam.transferPnPRightAxisX.pos02_vision.inPos;
   #statTonTime[410].TON(IN := #_w1 AND "Unit1.Em5.ControlNodes".transferPnPRight."step".transition1[410],
                         PT := T#100ms);
   IF #statTonTime[410].Q THEN
       "Unit1.Em5.ControlNodes".transferPnPRight.sequence.status.nextStep := #JOB_4_STEP_30;
   END_IF;
END_REGION

REGION Network 32: Step[430] : Transfer PP Right Y-Axis Vision Pos
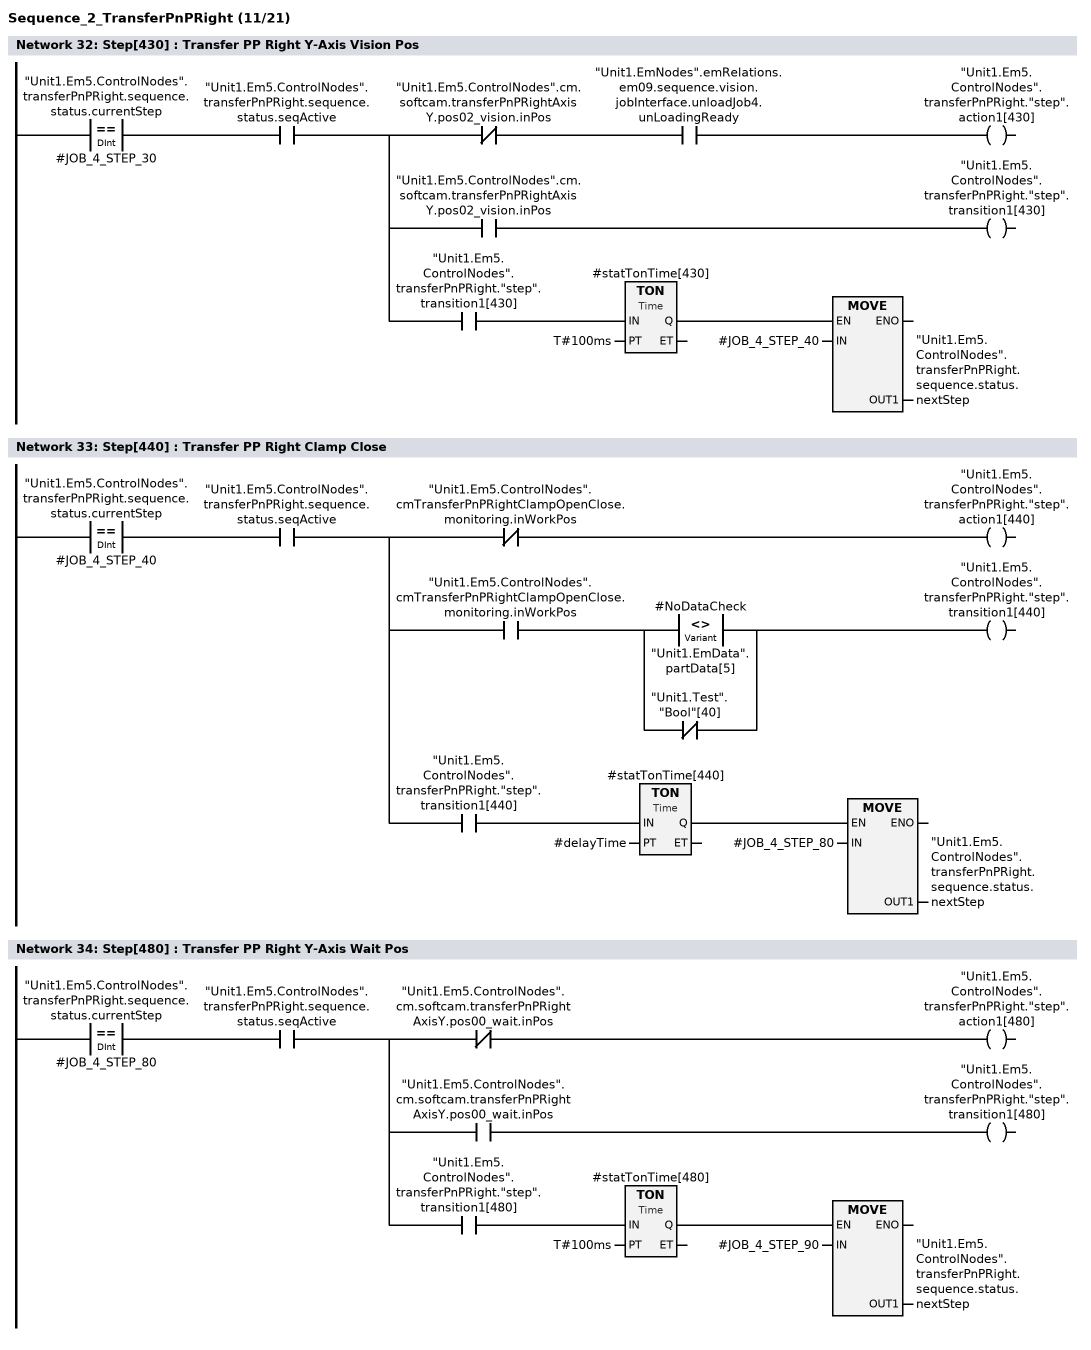
   RUNG wire#powerrail
      { S7_Templates := "SrcType := DInt" } EQ_Contact(in1 := "Unit1.Em5.ControlNodes".transferPnPRight.sequence.status.currentStep, in2 := #JOB_4_STEP_30)
      Contact( "Unit1.Em5.ControlNodes".transferPnPRight.sequence.status.seqActive )
      wire#w1
      I_Contact( "Unit1.Em5.ControlNodes".cm.softcam.transferPnPRightAxisY.pos02_vision.inPos )
      Contact( "Unit1.EmNodes".emRelations.em09.sequence.vision.jobInterface.unloadJob4.unLoadingReady )
      Coil( "Unit1.Em5.ControlNodes".transferPnPRight."step".action1[430] )
   END_RUNG
   RUNG wire#w1
      Contact( "Unit1.Em5.ControlNodes".cm.softcam.transferPnPRightAxisY.pos02_vision.inPos )
      Coil( "Unit1.Em5.ControlNodes".transferPnPRight."step".transition1[430] )
   END_RUNG
   RUNG wire#w1
      Contact( "Unit1.Em5.ControlNodes".transferPnPRight."step".transition1[430] )
      { S7_Templates := "time_type := Time" } #statTonTime[430].TON(pt := T#100ms, et =>)
      Move(in := #JOB_4_STEP_40, out1 => "Unit1.Em5.ControlNodes".transferPnPRight.sequence.status.nextStep)
   END_RUNG
   // the same network as SCL:
   #_w1 := ("Unit1.Em5.ControlNodes".transferPnPRight.sequence.status.currentStep = #JOB_4_STEP_30) AND "Unit1.Em5.ControlNodes".transferPnPRight.sequence.status.seqActive;
   "Unit1.Em5.ControlNodes".transferPnPRight."step".action1[430] := #_w1 AND NOT "Unit1.Em5.ControlNodes".cm.softcam.transferPnPRightAxisY.pos02_vision.inPos AND "Unit1.EmNodes".emRelations.em09.sequence.vision.jobInterface.unloadJob4.unLoadingReady;
   "Unit1.Em5.ControlNodes".transferPnPRight."step".transition1[430] := #_w1 AND "Unit1.Em5.ControlNodes".cm.softcam.transferPnPRightAxisY.pos02_vision.inPos;
   #statTonTime[430].TON(IN := #_w1 AND "Unit1.Em5.ControlNodes".transferPnPRight."step".transition1[430],
                         PT := T#100ms);
   IF #statTonTime[430].Q THEN
       "Unit1.Em5.ControlNodes".transferPnPRight.sequence.status.nextStep := #JOB_4_STEP_40;
   END_IF;
END_REGION

REGION Network 33: Step[440] : Transfer PP Right Clamp Close
   RUNG wire#powerrail
      { S7_Templates := "SrcType := DInt" } EQ_Contact(in1 := "Unit1.Em5.ControlNodes".transferPnPRight.sequence.status.currentStep, in2 := #JOB_4_STEP_40)
      Contact( "Unit1.Em5.ControlNodes".transferPnPRight.sequence.status.seqActive )
      wire#w1
      I_Contact( "Unit1.Em5.ControlNodes".cmTransferPnPRightClampOpenClose.monitoring.inWorkPos )
      Coil( "Unit1.Em5.ControlNodes".transferPnPRight."step".action1[440] )
   END_RUNG
   RUNG wire#w1
      Contact( "Unit1.Em5.ControlNodes".cmTransferPnPRightClampOpenClose.monitoring.inWorkPos )
      wire#w2
      { S7_Templates := "SrcType := Variant" } NE_Contact(in1 := #NoDataCheck, in2 := "Unit1.EmData".partData[5])
      wire#w3
      Coil( "Unit1.Em5.ControlNodes".transferPnPRight."step".transition1[440] )
   END_RUNG
   RUNG wire#w2
      I_Contact( "Unit1.Test"."Bool"[40] )
   END_RUNG wire#w3
   RUNG wire#w1
      Contact( "Unit1.Em5.ControlNodes".transferPnPRight."step".transition1[440] )
      { S7_Templates := "time_type := Time" } #statTonTime[440].TON(pt := #delayTime, et =>)
      Move(in := #JOB_4_STEP_80, out1 => "Unit1.Em5.ControlNodes".transferPnPRight.sequence.status.nextStep)
   END_RUNG
   // the same network as SCL:
   #_w1 := ("Unit1.Em5.ControlNodes".transferPnPRight.sequence.status.currentStep = #JOB_4_STEP_40) AND "Unit1.Em5.ControlNodes".transferPnPRight.sequence.status.seqActive;
   "Unit1.Em5.ControlNodes".transferPnPRight."step".action1[440] := #_w1 AND NOT "Unit1.Em5.ControlNodes".cmTransferPnPRightClampOpenClose.monitoring.inWorkPos;
   "Unit1.Em5.ControlNodes".transferPnPRight."step".transition1[440] := #_w1 AND "Unit1.Em5.ControlNodes".cmTransferPnPRightClampOpenClose.monitoring.inWorkPos AND ((#NoDataCheck <> "Unit1.EmData".partData[5]) OR NOT "Unit1.Test"."Bool"[40]);
   #statTonTime[440].TON(IN := #_w1 AND "Unit1.Em5.ControlNodes".transferPnPRight."step".transition1[440],
                         PT := #delayTime);
   IF #statTonTime[440].Q THEN
       "Unit1.Em5.ControlNodes".transferPnPRight.sequence.status.nextStep := #JOB_4_STEP_80;
   END_IF;
END_REGION

REGION Network 34: Step[480] : Transfer PP Right Y-Axis Wait Pos
   RUNG wire#powerrail
      { S7_Templates := "SrcType := DInt" } EQ_Contact(in1 := "Unit1.Em5.ControlNodes".transferPnPRight.sequence.status.currentStep, in2 := #JOB_4_STEP_80)
      Contact( "Unit1.Em5.ControlNodes".transferPnPRight.sequence.status.seqActive )
      wire#w1
      I_Contact( "Unit1.Em5.ControlNodes".cm.softcam.transferPnPRightAxisY.pos00_wait.inPos )
      Coil( "Unit1.Em5.ControlNodes".transferPnPRight."step".action1[480] )
   END_RUNG
   RUNG wire#w1
      Contact( "Unit1.Em5.ControlNodes".cm.softcam.transferPnPRightAxisY.pos00_wait.inPos )
      Coil( "Unit1.Em5.ControlNodes".transferPnPRight."step".transition1[480] )
   END_RUNG
   RUNG wire#w1
      Contact( "Unit1.Em5.ControlNodes".transferPnPRight."step".transition1[480] )
      { S7_Templates := "time_type := Time" } #statTonTime[480].TON(pt := T#100ms, et =>)
      Move(in := #JOB_4_STEP_90, out1 => "Unit1.Em5.ControlNodes".transferPnPRight.sequence.status.nextStep)
   END_RUNG
   // the same network as SCL:
   #_w1 := ("Unit1.Em5.ControlNodes".transferPnPRight.sequence.status.currentStep = #JOB_4_STEP_80) AND "Unit1.Em5.ControlNodes".transferPnPRight.sequence.status.seqActive;
   "Unit1.Em5.ControlNodes".transferPnPRight."step".action1[480] := #_w1 AND NOT "Unit1.Em5.ControlNodes".cm.softcam.transferPnPRightAxisY.pos00_wait.inPos;
   "Unit1.Em5.ControlNodes".transferPnPRight."step".transition1[480] := #_w1 AND "Unit1.Em5.ControlNodes".cm.softcam.transferPnPRightAxisY.pos00_wait.inPos;
   #statTonTime[480].TON(IN := #_w1 AND "Unit1.Em5.ControlNodes".transferPnPRight."step".transition1[480],
                         PT := T#100ms);
   IF #statTonTime[480].Q THEN
       "Unit1.Em5.ControlNodes".transferPnPRight.sequence.status.nextStep := #JOB_4_STEP_90;
   END_IF;
END_REGION

REGION Network 35: Step[490] : JOB[4] Step End
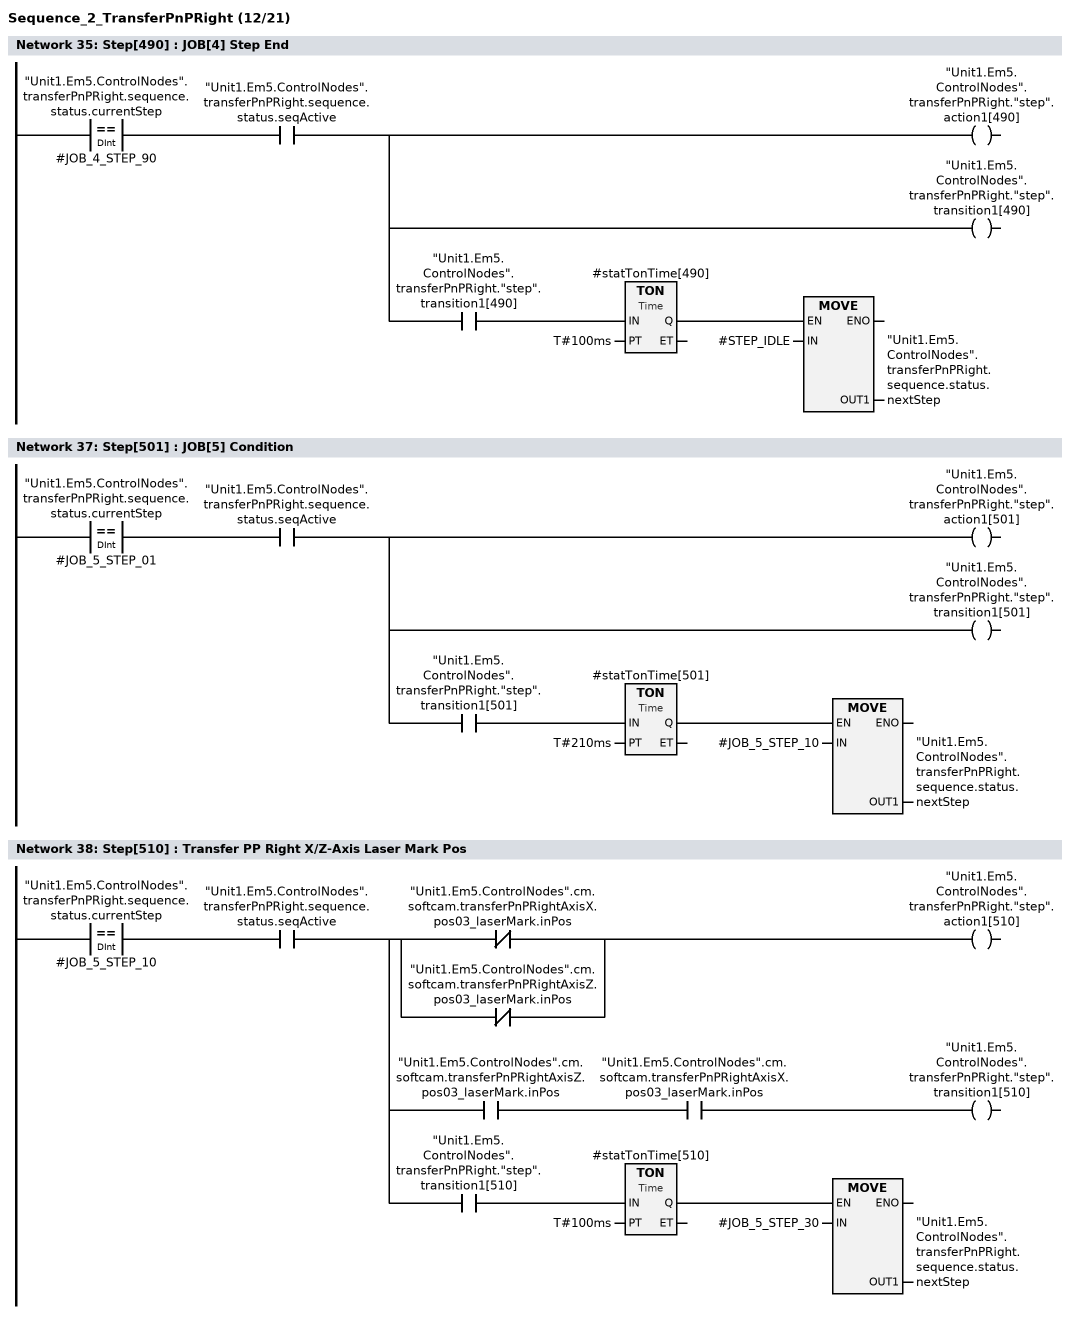
   RUNG wire#powerrail
      { S7_Templates := "SrcType := DInt" } EQ_Contact(in1 := "Unit1.Em5.ControlNodes".transferPnPRight.sequence.status.currentStep, in2 := #JOB_4_STEP_90)
      Contact( "Unit1.Em5.ControlNodes".transferPnPRight.sequence.status.seqActive )
      wire#w1
      Coil( "Unit1.Em5.ControlNodes".transferPnPRight."step".action1[490] )
   END_RUNG
   RUNG wire#w1
      Coil( "Unit1.Em5.ControlNodes".transferPnPRight."step".transition1[490] )
   END_RUNG
   RUNG wire#w1
      Contact( "Unit1.Em5.ControlNodes".transferPnPRight."step".transition1[490] )
      { S7_Templates := "time_type := Time" } #statTonTime[490].TON(pt := T#100ms, et =>)
      Move(in := #STEP_IDLE, out1 => "Unit1.Em5.ControlNodes".transferPnPRight.sequence.status.nextStep)
   END_RUNG
   // the same network as SCL:
   "Unit1.Em5.ControlNodes".transferPnPRight."step".action1[490] := ("Unit1.Em5.ControlNodes".transferPnPRight.sequence.status.currentStep = #JOB_4_STEP_90) AND "Unit1.Em5.ControlNodes".transferPnPRight.sequence.status.seqActive;
   "Unit1.Em5.ControlNodes".transferPnPRight."step".transition1[490] := ("Unit1.Em5.ControlNodes".transferPnPRight.sequence.status.currentStep = #JOB_4_STEP_90) AND "Unit1.Em5.ControlNodes".transferPnPRight.sequence.status.seqActive;
   #statTonTime[490].TON(IN := ("Unit1.Em5.ControlNodes".transferPnPRight.sequence.status.currentStep = #JOB_4_STEP_90) AND "Unit1.Em5.ControlNodes".transferPnPRight.sequence.status.seqActive AND "Unit1.Em5.ControlNodes".transferPnPRight."step".transition1[490],
                         PT := T#100ms);
   IF #statTonTime[490].Q THEN
       "Unit1.Em5.ControlNodes".transferPnPRight.sequence.status.nextStep := #STEP_IDLE;
   END_IF;
END_REGION

REGION Network 36: ************** JOB[5] LASER MARK JR PUT=AUTO-[A] ****************
END_REGION

REGION Network 37: Step[501] : JOB[5] Condition
   RUNG wire#powerrail
      { S7_Templates := "SrcType := DInt" } EQ_Contact(in1 := "Unit1.Em5.ControlNodes".transferPnPRight.sequence.status.currentStep, in2 := #JOB_5_STEP_01)
      Contact( "Unit1.Em5.ControlNodes".transferPnPRight.sequence.status.seqActive )
      wire#w1
      Coil( "Unit1.Em5.ControlNodes".transferPnPRight."step".action1[501] )
   END_RUNG
   RUNG wire#w1
      Coil( "Unit1.Em5.ControlNodes".transferPnPRight."step".transition1[501] )
   END_RUNG
   RUNG wire#w1
      Contact( "Unit1.Em5.ControlNodes".transferPnPRight."step".transition1[501] )
      { S7_Templates := "time_type := Time" } #statTonTime[501].TON(pt := T#210ms, et =>)
      Move(in := #JOB_5_STEP_10, out1 => "Unit1.Em5.ControlNodes".transferPnPRight.sequence.status.nextStep)
   END_RUNG
   // the same network as SCL:
   "Unit1.Em5.ControlNodes".transferPnPRight."step".action1[501] := ("Unit1.Em5.ControlNodes".transferPnPRight.sequence.status.currentStep = #JOB_5_STEP_01) AND "Unit1.Em5.ControlNodes".transferPnPRight.sequence.status.seqActive;
   "Unit1.Em5.ControlNodes".transferPnPRight."step".transition1[501] := ("Unit1.Em5.ControlNodes".transferPnPRight.sequence.status.currentStep = #JOB_5_STEP_01) AND "Unit1.Em5.ControlNodes".transferPnPRight.sequence.status.seqActive;
   #statTonTime[501].TON(IN := ("Unit1.Em5.ControlNodes".transferPnPRight.sequence.status.currentStep = #JOB_5_STEP_01) AND "Unit1.Em5.ControlNodes".transferPnPRight.sequence.status.seqActive AND "Unit1.Em5.ControlNodes".transferPnPRight."step".transition1[501],
                         PT := T#210ms);
   IF #statTonTime[501].Q THEN
       "Unit1.Em5.ControlNodes".transferPnPRight.sequence.status.nextStep := #JOB_5_STEP_10;
   END_IF;
END_REGION

REGION Network 38: Step[510] : Transfer PP Right X/Z-Axis Laser Mark Pos
   RUNG wire#powerrail
      { S7_Templates := "SrcType := DInt" } EQ_Contact(in1 := "Unit1.Em5.ControlNodes".transferPnPRight.sequence.status.currentStep, in2 := #JOB_5_STEP_10)
      Contact( "Unit1.Em5.ControlNodes".transferPnPRight.sequence.status.seqActive )
      wire#w1
      I_Contact( "Unit1.Em5.ControlNodes".cm.softcam.transferPnPRightAxisX.pos03_laserMark.inPos )
      wire#w2
      Coil( "Unit1.Em5.ControlNodes".transferPnPRight."step".action1[510] )
   END_RUNG
   RUNG wire#w1
      I_Contact( "Unit1.Em5.ControlNodes".cm.softcam.transferPnPRightAxisZ.pos03_laserMark.inPos )
   END_RUNG wire#w2
   RUNG wire#w1
      Contact( "Unit1.Em5.ControlNodes".cm.softcam.transferPnPRightAxisZ.pos03_laserMark.inPos )
      Contact( "Unit1.Em5.ControlNodes".cm.softcam.transferPnPRightAxisX.pos03_laserMark.inPos )
      Coil( "Unit1.Em5.ControlNodes".transferPnPRight."step".transition1[510] )
   END_RUNG
   RUNG wire#w1
      Contact( "Unit1.Em5.ControlNodes".transferPnPRight."step".transition1[510] )
      { S7_Templates := "time_type := Time" } #statTonTime[510].TON(pt := T#100ms, et =>)
      Move(in := #JOB_5_STEP_30, out1 => "Unit1.Em5.ControlNodes".transferPnPRight.sequence.status.nextStep)
   END_RUNG
   // the same network as SCL:
   #_w1 := ("Unit1.Em5.ControlNodes".transferPnPRight.sequence.status.currentStep = #JOB_5_STEP_10) AND "Unit1.Em5.ControlNodes".transferPnPRight.sequence.status.seqActive;
   "Unit1.Em5.ControlNodes".transferPnPRight."step".action1[510] := #_w1 AND (NOT "Unit1.Em5.ControlNodes".cm.softcam.transferPnPRightAxisX.pos03_laserMark.inPos OR NOT "Unit1.Em5.ControlNodes".cm.softcam.transferPnPRightAxisZ.pos03_laserMark.inPos);
   "Unit1.Em5.ControlNodes".transferPnPRight."step".transition1[510] := #_w1 AND "Unit1.Em5.ControlNodes".cm.softcam.transferPnPRightAxisZ.pos03_laserMark.inPos AND "Unit1.Em5.ControlNodes".cm.softcam.transferPnPRightAxisX.pos03_laserMark.inPos;
   #statTonTime[510].TON(IN := #_w1 AND "Unit1.Em5.ControlNodes".transferPnPRight."step".transition1[510],
                         PT := T#100ms);
   IF #statTonTime[510].Q THEN
       "Unit1.Em5.ControlNodes".transferPnPRight.sequence.status.nextStep := #JOB_5_STEP_30;
   END_IF;
END_REGION

REGION Network 39: Step[530] : Transfer PP Right Y-Axis Laser Mark Pos
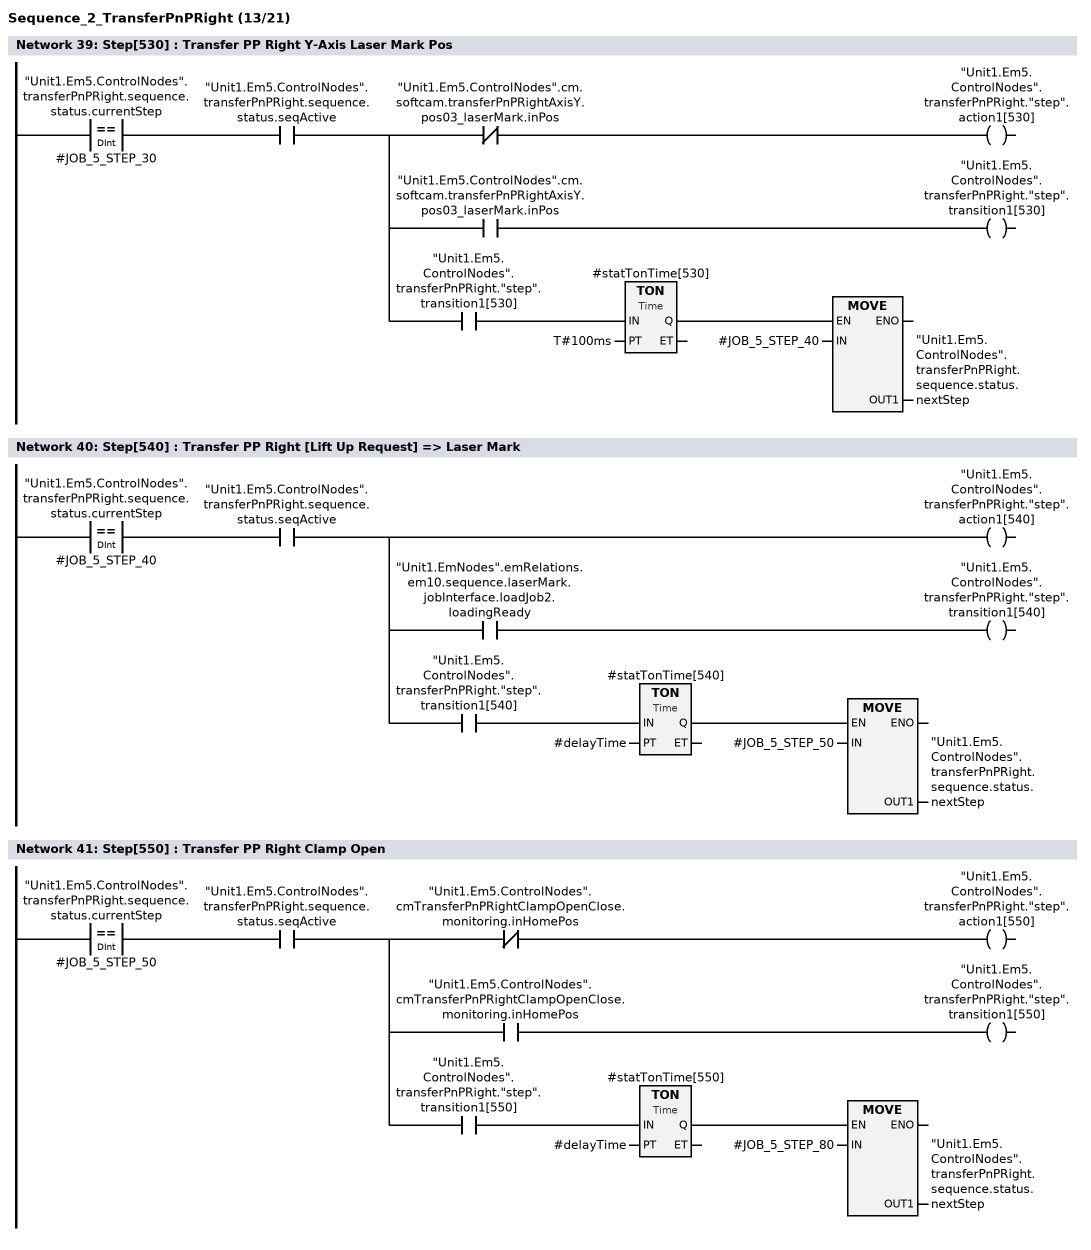
   RUNG wire#powerrail
      { S7_Templates := "SrcType := DInt" } EQ_Contact(in1 := "Unit1.Em5.ControlNodes".transferPnPRight.sequence.status.currentStep, in2 := #JOB_5_STEP_30)
      Contact( "Unit1.Em5.ControlNodes".transferPnPRight.sequence.status.seqActive )
      wire#w1
      I_Contact( "Unit1.Em5.ControlNodes".cm.softcam.transferPnPRightAxisY.pos03_laserMark.inPos )
      Coil( "Unit1.Em5.ControlNodes".transferPnPRight."step".action1[530] )
   END_RUNG
   RUNG wire#w1
      Contact( "Unit1.Em5.ControlNodes".cm.softcam.transferPnPRightAxisY.pos03_laserMark.inPos )
      Coil( "Unit1.Em5.ControlNodes".transferPnPRight."step".transition1[530] )
   END_RUNG
   RUNG wire#w1
      Contact( "Unit1.Em5.ControlNodes".transferPnPRight."step".transition1[530] )
      { S7_Templates := "time_type := Time" } #statTonTime[530].TON(pt := T#100ms, et =>)
      Move(in := #JOB_5_STEP_40, out1 => "Unit1.Em5.ControlNodes".transferPnPRight.sequence.status.nextStep)
   END_RUNG
   // the same network as SCL:
   #_w1 := ("Unit1.Em5.ControlNodes".transferPnPRight.sequence.status.currentStep = #JOB_5_STEP_30) AND "Unit1.Em5.ControlNodes".transferPnPRight.sequence.status.seqActive;
   "Unit1.Em5.ControlNodes".transferPnPRight."step".action1[530] := #_w1 AND NOT "Unit1.Em5.ControlNodes".cm.softcam.transferPnPRightAxisY.pos03_laserMark.inPos;
   "Unit1.Em5.ControlNodes".transferPnPRight."step".transition1[530] := #_w1 AND "Unit1.Em5.ControlNodes".cm.softcam.transferPnPRightAxisY.pos03_laserMark.inPos;
   #statTonTime[530].TON(IN := #_w1 AND "Unit1.Em5.ControlNodes".transferPnPRight."step".transition1[530],
                         PT := T#100ms);
   IF #statTonTime[530].Q THEN
       "Unit1.Em5.ControlNodes".transferPnPRight.sequence.status.nextStep := #JOB_5_STEP_40;
   END_IF;
END_REGION

REGION Network 40: Step[540] : Transfer PP Right [Lift Up Request] => Laser Mark
   RUNG wire#powerrail
      { S7_Templates := "SrcType := DInt" } EQ_Contact(in1 := "Unit1.Em5.ControlNodes".transferPnPRight.sequence.status.currentStep, in2 := #JOB_5_STEP_40)
      Contact( "Unit1.Em5.ControlNodes".transferPnPRight.sequence.status.seqActive )
      wire#w1
      Coil( "Unit1.Em5.ControlNodes".transferPnPRight."step".action1[540] )
   END_RUNG
   RUNG wire#w1
      Contact( "Unit1.EmNodes".emRelations.em10.sequence.laserMark.jobInterface.loadJob2.loadingReady )
      Coil( "Unit1.Em5.ControlNodes".transferPnPRight."step".transition1[540] )
   END_RUNG
   RUNG wire#w1
      Contact( "Unit1.Em5.ControlNodes".transferPnPRight."step".transition1[540] )
      { S7_Templates := "time_type := Time" } #statTonTime[540].TON(pt := #delayTime, et =>)
      Move(in := #JOB_5_STEP_50, out1 => "Unit1.Em5.ControlNodes".transferPnPRight.sequence.status.nextStep)
   END_RUNG
   // the same network as SCL:
   "Unit1.Em5.ControlNodes".transferPnPRight."step".action1[540] := ("Unit1.Em5.ControlNodes".transferPnPRight.sequence.status.currentStep = #JOB_5_STEP_40) AND "Unit1.Em5.ControlNodes".transferPnPRight.sequence.status.seqActive;
   "Unit1.Em5.ControlNodes".transferPnPRight."step".transition1[540] := ("Unit1.Em5.ControlNodes".transferPnPRight.sequence.status.currentStep = #JOB_5_STEP_40) AND "Unit1.Em5.ControlNodes".transferPnPRight.sequence.status.seqActive AND "Unit1.EmNodes".emRelations.em10.sequence.laserMark.jobInterface.loadJob2.loadingReady;
   #statTonTime[540].TON(IN := ("Unit1.Em5.ControlNodes".transferPnPRight.sequence.status.currentStep = #JOB_5_STEP_40) AND "Unit1.Em5.ControlNodes".transferPnPRight.sequence.status.seqActive AND "Unit1.Em5.ControlNodes".transferPnPRight."step".transition1[540],
                         PT := #delayTime);
   IF #statTonTime[540].Q THEN
       "Unit1.Em5.ControlNodes".transferPnPRight.sequence.status.nextStep := #JOB_5_STEP_50;
   END_IF;
END_REGION

REGION Network 41: Step[550] : Transfer PP Right Clamp Open
   RUNG wire#powerrail
      { S7_Templates := "SrcType := DInt" } EQ_Contact(in1 := "Unit1.Em5.ControlNodes".transferPnPRight.sequence.status.currentStep, in2 := #JOB_5_STEP_50)
      Contact( "Unit1.Em5.ControlNodes".transferPnPRight.sequence.status.seqActive )
      wire#w1
      I_Contact( "Unit1.Em5.ControlNodes".cmTransferPnPRightClampOpenClose.monitoring.inHomePos )
      Coil( "Unit1.Em5.ControlNodes".transferPnPRight."step".action1[550] )
   END_RUNG
   RUNG wire#w1
      Contact( "Unit1.Em5.ControlNodes".cmTransferPnPRightClampOpenClose.monitoring.inHomePos )
      Coil( "Unit1.Em5.ControlNodes".transferPnPRight."step".transition1[550] )
   END_RUNG
   RUNG wire#w1
      Contact( "Unit1.Em5.ControlNodes".transferPnPRight."step".transition1[550] )
      { S7_Templates := "time_type := Time" } #statTonTime[550].TON(pt := #delayTime, et =>)
      Move(in := #JOB_5_STEP_80, out1 => "Unit1.Em5.ControlNodes".transferPnPRight.sequence.status.nextStep)
   END_RUNG
   // the same network as SCL:
   #_w1 := ("Unit1.Em5.ControlNodes".transferPnPRight.sequence.status.currentStep = #JOB_5_STEP_50) AND "Unit1.Em5.ControlNodes".transferPnPRight.sequence.status.seqActive;
   "Unit1.Em5.ControlNodes".transferPnPRight."step".action1[550] := #_w1 AND NOT "Unit1.Em5.ControlNodes".cmTransferPnPRightClampOpenClose.monitoring.inHomePos;
   "Unit1.Em5.ControlNodes".transferPnPRight."step".transition1[550] := #_w1 AND "Unit1.Em5.ControlNodes".cmTransferPnPRightClampOpenClose.monitoring.inHomePos;
   #statTonTime[550].TON(IN := #_w1 AND "Unit1.Em5.ControlNodes".transferPnPRight."step".transition1[550],
                         PT := #delayTime);
   IF #statTonTime[550].Q THEN
       "Unit1.Em5.ControlNodes".transferPnPRight.sequence.status.nextStep := #JOB_5_STEP_80;
   END_IF;
END_REGION

REGION Network 42: Step[580] : Transfer PP Right Y-Axis Wait Pos
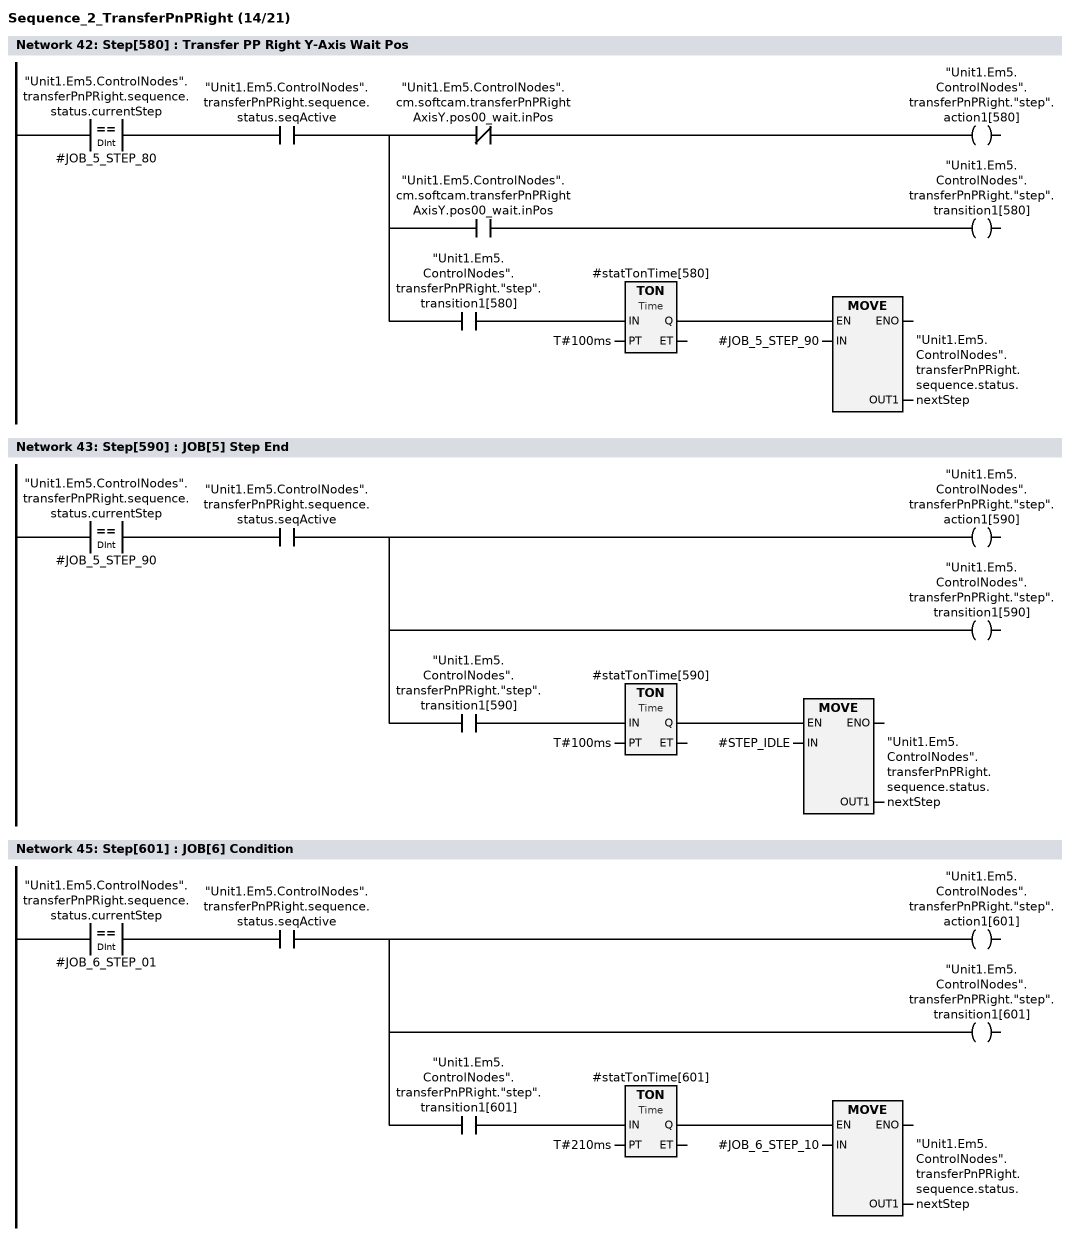
   RUNG wire#powerrail
      { S7_Templates := "SrcType := DInt" } EQ_Contact(in1 := "Unit1.Em5.ControlNodes".transferPnPRight.sequence.status.currentStep, in2 := #JOB_5_STEP_80)
      Contact( "Unit1.Em5.ControlNodes".transferPnPRight.sequence.status.seqActive )
      wire#w1
      I_Contact( "Unit1.Em5.ControlNodes".cm.softcam.transferPnPRightAxisY.pos00_wait.inPos )
      Coil( "Unit1.Em5.ControlNodes".transferPnPRight."step".action1[580] )
   END_RUNG
   RUNG wire#w1
      Contact( "Unit1.Em5.ControlNodes".cm.softcam.transferPnPRightAxisY.pos00_wait.inPos )
      Coil( "Unit1.Em5.ControlNodes".transferPnPRight."step".transition1[580] )
   END_RUNG
   RUNG wire#w1
      Contact( "Unit1.Em5.ControlNodes".transferPnPRight."step".transition1[580] )
      { S7_Templates := "time_type := Time" } #statTonTime[580].TON(pt := T#100ms, et =>)
      Move(in := #JOB_5_STEP_90, out1 => "Unit1.Em5.ControlNodes".transferPnPRight.sequence.status.nextStep)
   END_RUNG
   // the same network as SCL:
   #_w1 := ("Unit1.Em5.ControlNodes".transferPnPRight.sequence.status.currentStep = #JOB_5_STEP_80) AND "Unit1.Em5.ControlNodes".transferPnPRight.sequence.status.seqActive;
   "Unit1.Em5.ControlNodes".transferPnPRight."step".action1[580] := #_w1 AND NOT "Unit1.Em5.ControlNodes".cm.softcam.transferPnPRightAxisY.pos00_wait.inPos;
   "Unit1.Em5.ControlNodes".transferPnPRight."step".transition1[580] := #_w1 AND "Unit1.Em5.ControlNodes".cm.softcam.transferPnPRightAxisY.pos00_wait.inPos;
   #statTonTime[580].TON(IN := #_w1 AND "Unit1.Em5.ControlNodes".transferPnPRight."step".transition1[580],
                         PT := T#100ms);
   IF #statTonTime[580].Q THEN
       "Unit1.Em5.ControlNodes".transferPnPRight.sequence.status.nextStep := #JOB_5_STEP_90;
   END_IF;
END_REGION

REGION Network 43: Step[590] : JOB[5] Step End
   RUNG wire#powerrail
      { S7_Templates := "SrcType := DInt" } EQ_Contact(in1 := "Unit1.Em5.ControlNodes".transferPnPRight.sequence.status.currentStep, in2 := #JOB_5_STEP_90)
      Contact( "Unit1.Em5.ControlNodes".transferPnPRight.sequence.status.seqActive )
      wire#w1
      Coil( "Unit1.Em5.ControlNodes".transferPnPRight."step".action1[590] )
   END_RUNG
   RUNG wire#w1
      Coil( "Unit1.Em5.ControlNodes".transferPnPRight."step".transition1[590] )
   END_RUNG
   RUNG wire#w1
      Contact( "Unit1.Em5.ControlNodes".transferPnPRight."step".transition1[590] )
      { S7_Templates := "time_type := Time" } #statTonTime[590].TON(pt := T#100ms, et =>)
      Move(in := #STEP_IDLE, out1 => "Unit1.Em5.ControlNodes".transferPnPRight.sequence.status.nextStep)
   END_RUNG
   // the same network as SCL:
   "Unit1.Em5.ControlNodes".transferPnPRight."step".action1[590] := ("Unit1.Em5.ControlNodes".transferPnPRight.sequence.status.currentStep = #JOB_5_STEP_90) AND "Unit1.Em5.ControlNodes".transferPnPRight.sequence.status.seqActive;
   "Unit1.Em5.ControlNodes".transferPnPRight."step".transition1[590] := ("Unit1.Em5.ControlNodes".transferPnPRight.sequence.status.currentStep = #JOB_5_STEP_90) AND "Unit1.Em5.ControlNodes".transferPnPRight.sequence.status.seqActive;
   #statTonTime[590].TON(IN := ("Unit1.Em5.ControlNodes".transferPnPRight.sequence.status.currentStep = #JOB_5_STEP_90) AND "Unit1.Em5.ControlNodes".transferPnPRight.sequence.status.seqActive AND "Unit1.Em5.ControlNodes".transferPnPRight."step".transition1[590],
                         PT := T#100ms);
   IF #statTonTime[590].Q THEN
       "Unit1.Em5.ControlNodes".transferPnPRight.sequence.status.nextStep := #STEP_IDLE;
   END_IF;
END_REGION

REGION Network 44: ************** JOB[6] LASER MARK JR GET=AUTO-[A] ****************
END_REGION

REGION Network 45: Step[601] : JOB[6] Condition
   RUNG wire#powerrail
      { S7_Templates := "SrcType := DInt" } EQ_Contact(in1 := "Unit1.Em5.ControlNodes".transferPnPRight.sequence.status.currentStep, in2 := #JOB_6_STEP_01)
      Contact( "Unit1.Em5.ControlNodes".transferPnPRight.sequence.status.seqActive )
      wire#w1
      Coil( "Unit1.Em5.ControlNodes".transferPnPRight."step".action1[601] )
   END_RUNG
   RUNG wire#w1
      Coil( "Unit1.Em5.ControlNodes".transferPnPRight."step".transition1[601] )
   END_RUNG
   RUNG wire#w1
      Contact( "Unit1.Em5.ControlNodes".transferPnPRight."step".transition1[601] )
      { S7_Templates := "time_type := Time" } #statTonTime[601].TON(pt := T#210ms, et =>)
      Move(in := #JOB_6_STEP_10, out1 => "Unit1.Em5.ControlNodes".transferPnPRight.sequence.status.nextStep)
   END_RUNG
   // the same network as SCL:
   "Unit1.Em5.ControlNodes".transferPnPRight."step".action1[601] := ("Unit1.Em5.ControlNodes".transferPnPRight.sequence.status.currentStep = #JOB_6_STEP_01) AND "Unit1.Em5.ControlNodes".transferPnPRight.sequence.status.seqActive;
   "Unit1.Em5.ControlNodes".transferPnPRight."step".transition1[601] := ("Unit1.Em5.ControlNodes".transferPnPRight.sequence.status.currentStep = #JOB_6_STEP_01) AND "Unit1.Em5.ControlNodes".transferPnPRight.sequence.status.seqActive;
   #statTonTime[601].TON(IN := ("Unit1.Em5.ControlNodes".transferPnPRight.sequence.status.currentStep = #JOB_6_STEP_01) AND "Unit1.Em5.ControlNodes".transferPnPRight.sequence.status.seqActive AND "Unit1.Em5.ControlNodes".transferPnPRight."step".transition1[601],
                         PT := T#210ms);
   IF #statTonTime[601].Q THEN
       "Unit1.Em5.ControlNodes".transferPnPRight.sequence.status.nextStep := #JOB_6_STEP_10;
   END_IF;
END_REGION

REGION Network 46: Step[610] : Transfer PP Right X/Z-Axis Laser Mark Pos
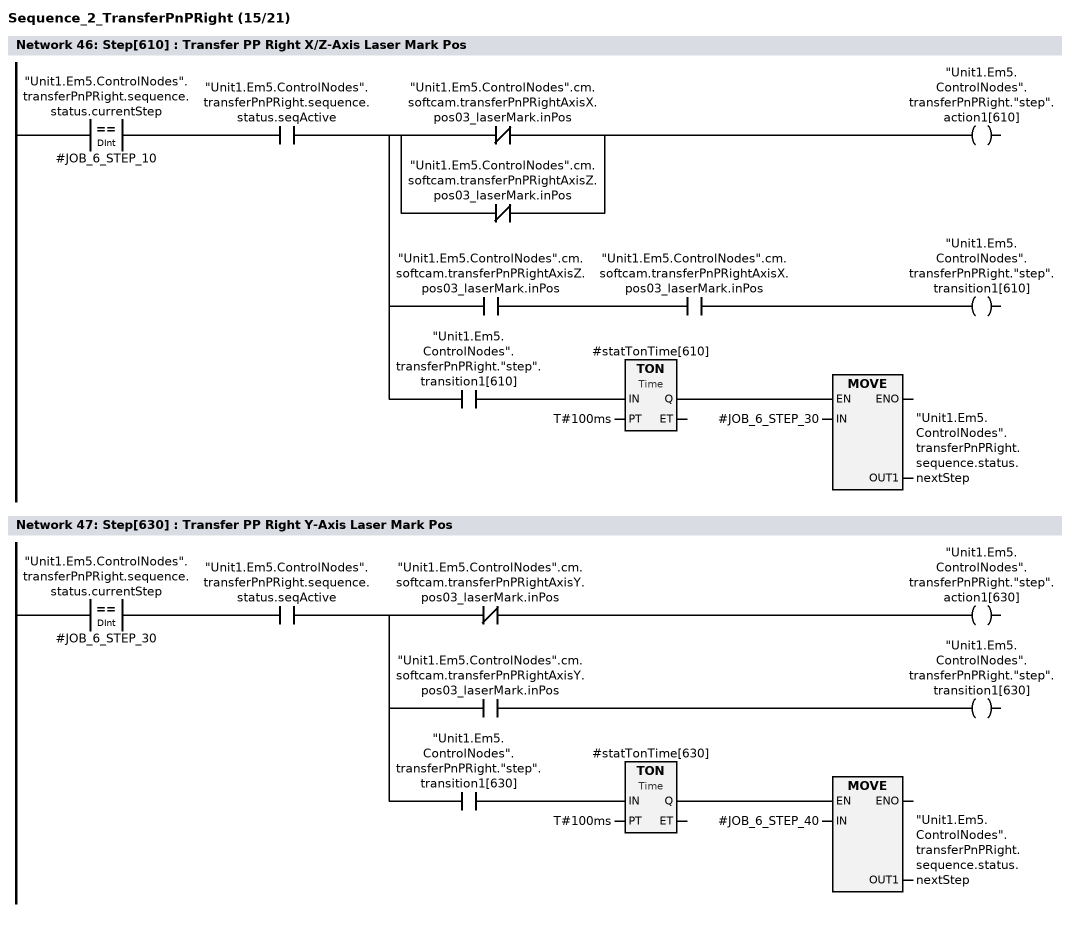
   RUNG wire#powerrail
      { S7_Templates := "SrcType := DInt" } EQ_Contact(in1 := "Unit1.Em5.ControlNodes".transferPnPRight.sequence.status.currentStep, in2 := #JOB_6_STEP_10)
      Contact( "Unit1.Em5.ControlNodes".transferPnPRight.sequence.status.seqActive )
      wire#w1
      I_Contact( "Unit1.Em5.ControlNodes".cm.softcam.transferPnPRightAxisX.pos03_laserMark.inPos )
      wire#w2
      Coil( "Unit1.Em5.ControlNodes".transferPnPRight."step".action1[610] )
   END_RUNG
   RUNG wire#w1
      I_Contact( "Unit1.Em5.ControlNodes".cm.softcam.transferPnPRightAxisZ.pos03_laserMark.inPos )
   END_RUNG wire#w2
   RUNG wire#w1
      Contact( "Unit1.Em5.ControlNodes".cm.softcam.transferPnPRightAxisZ.pos03_laserMark.inPos )
      Contact( "Unit1.Em5.ControlNodes".cm.softcam.transferPnPRightAxisX.pos03_laserMark.inPos )
      Coil( "Unit1.Em5.ControlNodes".transferPnPRight."step".transition1[610] )
   END_RUNG
   RUNG wire#w1
      Contact( "Unit1.Em5.ControlNodes".transferPnPRight."step".transition1[610] )
      { S7_Templates := "time_type := Time" } #statTonTime[610].TON(pt := T#100ms, et =>)
      Move(in := #JOB_6_STEP_30, out1 => "Unit1.Em5.ControlNodes".transferPnPRight.sequence.status.nextStep)
   END_RUNG
   // the same network as SCL:
   #_w1 := ("Unit1.Em5.ControlNodes".transferPnPRight.sequence.status.currentStep = #JOB_6_STEP_10) AND "Unit1.Em5.ControlNodes".transferPnPRight.sequence.status.seqActive;
   "Unit1.Em5.ControlNodes".transferPnPRight."step".action1[610] := #_w1 AND (NOT "Unit1.Em5.ControlNodes".cm.softcam.transferPnPRightAxisX.pos03_laserMark.inPos OR NOT "Unit1.Em5.ControlNodes".cm.softcam.transferPnPRightAxisZ.pos03_laserMark.inPos);
   "Unit1.Em5.ControlNodes".transferPnPRight."step".transition1[610] := #_w1 AND "Unit1.Em5.ControlNodes".cm.softcam.transferPnPRightAxisZ.pos03_laserMark.inPos AND "Unit1.Em5.ControlNodes".cm.softcam.transferPnPRightAxisX.pos03_laserMark.inPos;
   #statTonTime[610].TON(IN := #_w1 AND "Unit1.Em5.ControlNodes".transferPnPRight."step".transition1[610],
                         PT := T#100ms);
   IF #statTonTime[610].Q THEN
       "Unit1.Em5.ControlNodes".transferPnPRight.sequence.status.nextStep := #JOB_6_STEP_30;
   END_IF;
END_REGION

REGION Network 47: Step[630] : Transfer PP Right Y-Axis Laser Mark Pos
   RUNG wire#powerrail
      { S7_Templates := "SrcType := DInt" } EQ_Contact(in1 := "Unit1.Em5.ControlNodes".transferPnPRight.sequence.status.currentStep, in2 := #JOB_6_STEP_30)
      Contact( "Unit1.Em5.ControlNodes".transferPnPRight.sequence.status.seqActive )
      wire#w1
      I_Contact( "Unit1.Em5.ControlNodes".cm.softcam.transferPnPRightAxisY.pos03_laserMark.inPos )
      Coil( "Unit1.Em5.ControlNodes".transferPnPRight."step".action1[630] )
   END_RUNG
   RUNG wire#w1
      Contact( "Unit1.Em5.ControlNodes".cm.softcam.transferPnPRightAxisY.pos03_laserMark.inPos )
      Coil( "Unit1.Em5.ControlNodes".transferPnPRight."step".transition1[630] )
   END_RUNG
   RUNG wire#w1
      Contact( "Unit1.Em5.ControlNodes".transferPnPRight."step".transition1[630] )
      { S7_Templates := "time_type := Time" } #statTonTime[630].TON(pt := T#100ms, et =>)
      Move(in := #JOB_6_STEP_40, out1 => "Unit1.Em5.ControlNodes".transferPnPRight.sequence.status.nextStep)
   END_RUNG
   // the same network as SCL:
   #_w1 := ("Unit1.Em5.ControlNodes".transferPnPRight.sequence.status.currentStep = #JOB_6_STEP_30) AND "Unit1.Em5.ControlNodes".transferPnPRight.sequence.status.seqActive;
   "Unit1.Em5.ControlNodes".transferPnPRight."step".action1[630] := #_w1 AND NOT "Unit1.Em5.ControlNodes".cm.softcam.transferPnPRightAxisY.pos03_laserMark.inPos;
   "Unit1.Em5.ControlNodes".transferPnPRight."step".transition1[630] := #_w1 AND "Unit1.Em5.ControlNodes".cm.softcam.transferPnPRightAxisY.pos03_laserMark.inPos;
   #statTonTime[630].TON(IN := #_w1 AND "Unit1.Em5.ControlNodes".transferPnPRight."step".transition1[630],
                         PT := T#100ms);
   IF #statTonTime[630].Q THEN
       "Unit1.Em5.ControlNodes".transferPnPRight.sequence.status.nextStep := #JOB_6_STEP_40;
   END_IF;
END_REGION

REGION Network 48: Step[640] : Transfer PP Right Clamp Close
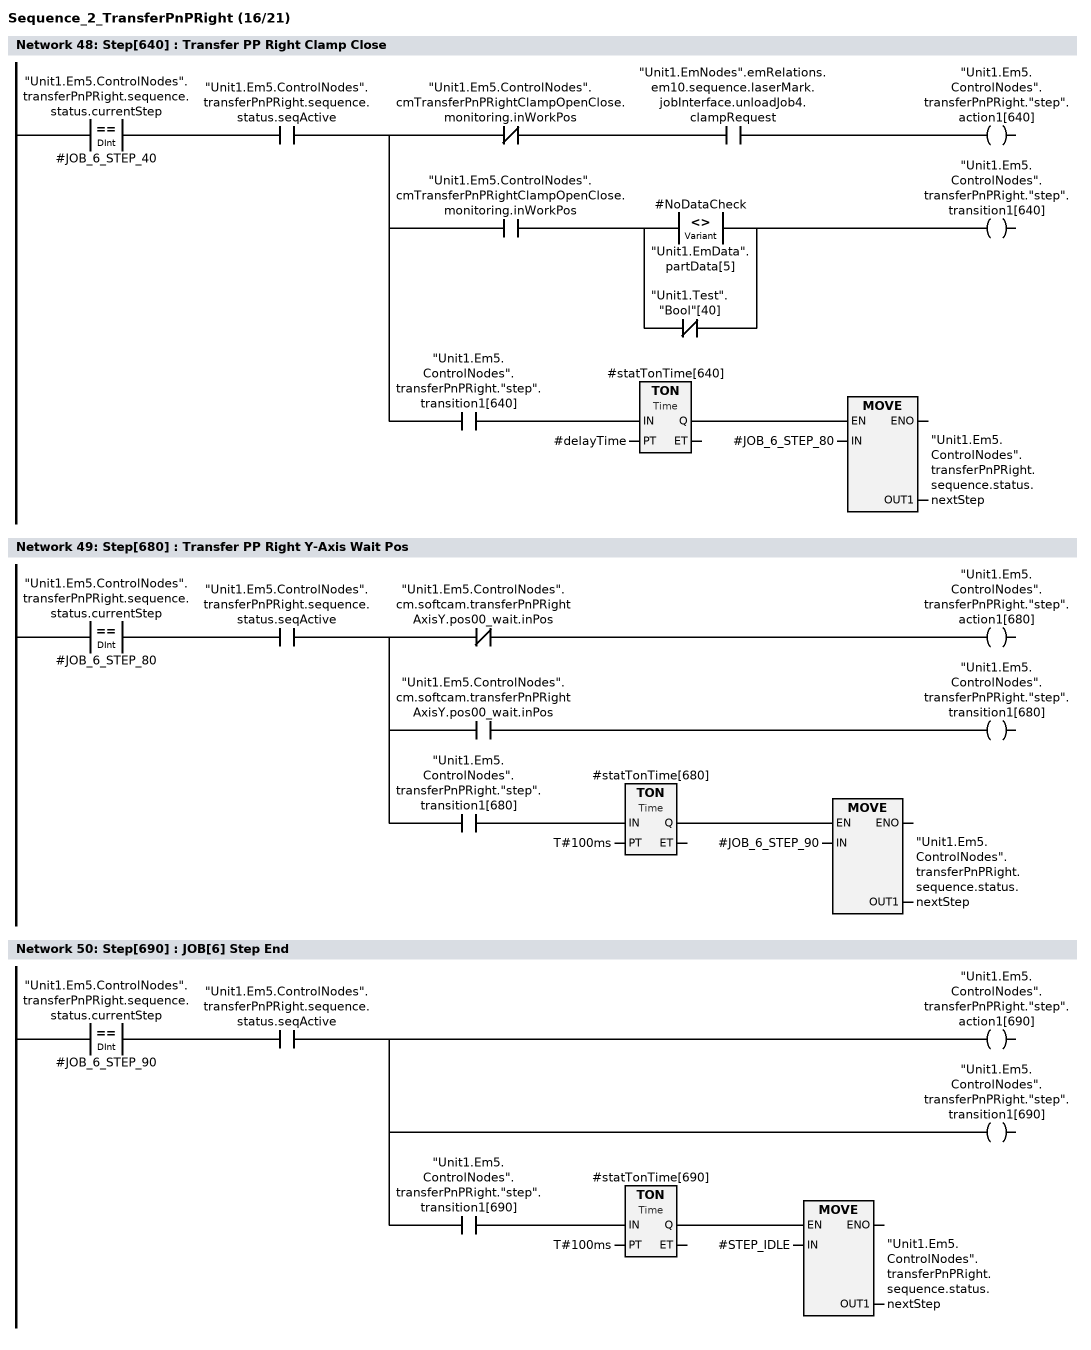
   RUNG wire#powerrail
      { S7_Templates := "SrcType := DInt" } EQ_Contact(in1 := "Unit1.Em5.ControlNodes".transferPnPRight.sequence.status.currentStep, in2 := #JOB_6_STEP_40)
      Contact( "Unit1.Em5.ControlNodes".transferPnPRight.sequence.status.seqActive )
      wire#w1
      I_Contact( "Unit1.Em5.ControlNodes".cmTransferPnPRightClampOpenClose.monitoring.inWorkPos )
      Contact( "Unit1.EmNodes".emRelations.em10.sequence.laserMark.jobInterface.unloadJob4.clampRequest )
      Coil( "Unit1.Em5.ControlNodes".transferPnPRight."step".action1[640] )
   END_RUNG
   RUNG wire#w1
      Contact( "Unit1.Em5.ControlNodes".cmTransferPnPRightClampOpenClose.monitoring.inWorkPos )
      wire#w2
      { S7_Templates := "SrcType := Variant" } NE_Contact(in1 := #NoDataCheck, in2 := "Unit1.EmData".partData[5])
      wire#w3
      Coil( "Unit1.Em5.ControlNodes".transferPnPRight."step".transition1[640] )
   END_RUNG
   RUNG wire#w2
      I_Contact( "Unit1.Test"."Bool"[40] )
   END_RUNG wire#w3
   RUNG wire#w1
      Contact( "Unit1.Em5.ControlNodes".transferPnPRight."step".transition1[640] )
      { S7_Templates := "time_type := Time" } #statTonTime[640].TON(pt := #delayTime, et =>)
      Move(in := #JOB_6_STEP_80, out1 => "Unit1.Em5.ControlNodes".transferPnPRight.sequence.status.nextStep)
   END_RUNG
   // the same network as SCL:
   #_w1 := ("Unit1.Em5.ControlNodes".transferPnPRight.sequence.status.currentStep = #JOB_6_STEP_40) AND "Unit1.Em5.ControlNodes".transferPnPRight.sequence.status.seqActive;
   "Unit1.Em5.ControlNodes".transferPnPRight."step".action1[640] := #_w1 AND NOT "Unit1.Em5.ControlNodes".cmTransferPnPRightClampOpenClose.monitoring.inWorkPos AND "Unit1.EmNodes".emRelations.em10.sequence.laserMark.jobInterface.unloadJob4.clampRequest;
   "Unit1.Em5.ControlNodes".transferPnPRight."step".transition1[640] := #_w1 AND "Unit1.Em5.ControlNodes".cmTransferPnPRightClampOpenClose.monitoring.inWorkPos AND ((#NoDataCheck <> "Unit1.EmData".partData[5]) OR NOT "Unit1.Test"."Bool"[40]);
   #statTonTime[640].TON(IN := #_w1 AND "Unit1.Em5.ControlNodes".transferPnPRight."step".transition1[640],
                         PT := #delayTime);
   IF #statTonTime[640].Q THEN
       "Unit1.Em5.ControlNodes".transferPnPRight.sequence.status.nextStep := #JOB_6_STEP_80;
   END_IF;
END_REGION

REGION Network 49: Step[680] : Transfer PP Right Y-Axis Wait Pos
   RUNG wire#powerrail
      { S7_Templates := "SrcType := DInt" } EQ_Contact(in1 := "Unit1.Em5.ControlNodes".transferPnPRight.sequence.status.currentStep, in2 := #JOB_6_STEP_80)
      Contact( "Unit1.Em5.ControlNodes".transferPnPRight.sequence.status.seqActive )
      wire#w1
      I_Contact( "Unit1.Em5.ControlNodes".cm.softcam.transferPnPRightAxisY.pos00_wait.inPos )
      Coil( "Unit1.Em5.ControlNodes".transferPnPRight."step".action1[680] )
   END_RUNG
   RUNG wire#w1
      Contact( "Unit1.Em5.ControlNodes".cm.softcam.transferPnPRightAxisY.pos00_wait.inPos )
      Coil( "Unit1.Em5.ControlNodes".transferPnPRight."step".transition1[680] )
   END_RUNG
   RUNG wire#w1
      Contact( "Unit1.Em5.ControlNodes".transferPnPRight."step".transition1[680] )
      { S7_Templates := "time_type := Time" } #statTonTime[680].TON(pt := T#100ms, et =>)
      Move(in := #JOB_6_STEP_90, out1 => "Unit1.Em5.ControlNodes".transferPnPRight.sequence.status.nextStep)
   END_RUNG
   // the same network as SCL:
   #_w1 := ("Unit1.Em5.ControlNodes".transferPnPRight.sequence.status.currentStep = #JOB_6_STEP_80) AND "Unit1.Em5.ControlNodes".transferPnPRight.sequence.status.seqActive;
   "Unit1.Em5.ControlNodes".transferPnPRight."step".action1[680] := #_w1 AND NOT "Unit1.Em5.ControlNodes".cm.softcam.transferPnPRightAxisY.pos00_wait.inPos;
   "Unit1.Em5.ControlNodes".transferPnPRight."step".transition1[680] := #_w1 AND "Unit1.Em5.ControlNodes".cm.softcam.transferPnPRightAxisY.pos00_wait.inPos;
   #statTonTime[680].TON(IN := #_w1 AND "Unit1.Em5.ControlNodes".transferPnPRight."step".transition1[680],
                         PT := T#100ms);
   IF #statTonTime[680].Q THEN
       "Unit1.Em5.ControlNodes".transferPnPRight.sequence.status.nextStep := #JOB_6_STEP_90;
   END_IF;
END_REGION

REGION Network 50: Step[690] : JOB[6] Step End
   RUNG wire#powerrail
      { S7_Templates := "SrcType := DInt" } EQ_Contact(in1 := "Unit1.Em5.ControlNodes".transferPnPRight.sequence.status.currentStep, in2 := #JOB_6_STEP_90)
      Contact( "Unit1.Em5.ControlNodes".transferPnPRight.sequence.status.seqActive )
      wire#w1
      Coil( "Unit1.Em5.ControlNodes".transferPnPRight."step".action1[690] )
   END_RUNG
   RUNG wire#w1
      Coil( "Unit1.Em5.ControlNodes".transferPnPRight."step".transition1[690] )
   END_RUNG
   RUNG wire#w1
      Contact( "Unit1.Em5.ControlNodes".transferPnPRight."step".transition1[690] )
      { S7_Templates := "time_type := Time" } #statTonTime[690].TON(pt := T#100ms, et =>)
      Move(in := #STEP_IDLE, out1 => "Unit1.Em5.ControlNodes".transferPnPRight.sequence.status.nextStep)
   END_RUNG
   // the same network as SCL:
   "Unit1.Em5.ControlNodes".transferPnPRight."step".action1[690] := ("Unit1.Em5.ControlNodes".transferPnPRight.sequence.status.currentStep = #JOB_6_STEP_90) AND "Unit1.Em5.ControlNodes".transferPnPRight.sequence.status.seqActive;
   "Unit1.Em5.ControlNodes".transferPnPRight."step".transition1[690] := ("Unit1.Em5.ControlNodes".transferPnPRight.sequence.status.currentStep = #JOB_6_STEP_90) AND "Unit1.Em5.ControlNodes".transferPnPRight.sequence.status.seqActive;
   #statTonTime[690].TON(IN := ("Unit1.Em5.ControlNodes".transferPnPRight.sequence.status.currentStep = #JOB_6_STEP_90) AND "Unit1.Em5.ControlNodes".transferPnPRight.sequence.status.seqActive AND "Unit1.Em5.ControlNodes".transferPnPRight."step".transition1[690],
                         PT := T#100ms);
   IF #statTonTime[690].Q THEN
       "Unit1.Em5.ControlNodes".transferPnPRight.sequence.status.nextStep := #STEP_IDLE;
   END_IF;
END_REGION

REGION Network 51: ************* JOB[9] WEIGHT CHECK JR PUT=AUTO-[A][B] ****************
END_REGION

REGION Network 52: Step[901] : JOB[9] Condition
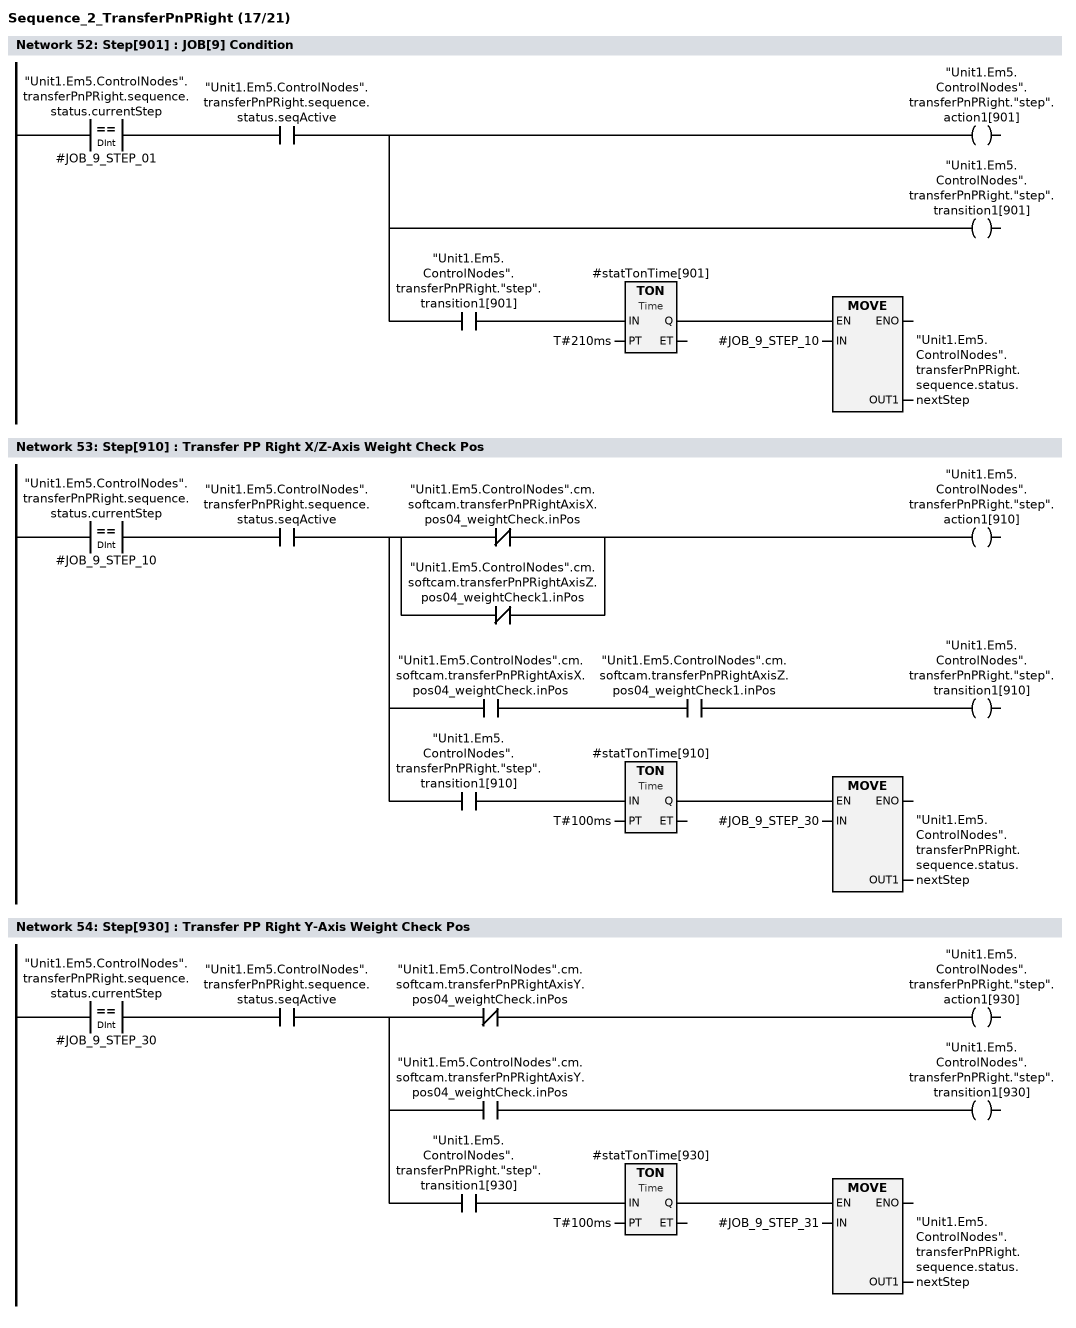
   RUNG wire#powerrail
      { S7_Templates := "SrcType := DInt" } EQ_Contact(in1 := "Unit1.Em5.ControlNodes".transferPnPRight.sequence.status.currentStep, in2 := #JOB_9_STEP_01)
      Contact( "Unit1.Em5.ControlNodes".transferPnPRight.sequence.status.seqActive )
      wire#w1
      Coil( "Unit1.Em5.ControlNodes".transferPnPRight."step".action1[901] )
   END_RUNG
   RUNG wire#w1
      Coil( "Unit1.Em5.ControlNodes".transferPnPRight."step".transition1[901] )
   END_RUNG
   RUNG wire#w1
      Contact( "Unit1.Em5.ControlNodes".transferPnPRight."step".transition1[901] )
      { S7_Templates := "time_type := Time" } #statTonTime[901].TON(pt := T#210ms, et =>)
      Move(in := #JOB_9_STEP_10, out1 => "Unit1.Em5.ControlNodes".transferPnPRight.sequence.status.nextStep)
   END_RUNG
   // the same network as SCL:
   "Unit1.Em5.ControlNodes".transferPnPRight."step".action1[901] := ("Unit1.Em5.ControlNodes".transferPnPRight.sequence.status.currentStep = #JOB_9_STEP_01) AND "Unit1.Em5.ControlNodes".transferPnPRight.sequence.status.seqActive;
   "Unit1.Em5.ControlNodes".transferPnPRight."step".transition1[901] := ("Unit1.Em5.ControlNodes".transferPnPRight.sequence.status.currentStep = #JOB_9_STEP_01) AND "Unit1.Em5.ControlNodes".transferPnPRight.sequence.status.seqActive;
   #statTonTime[901].TON(IN := ("Unit1.Em5.ControlNodes".transferPnPRight.sequence.status.currentStep = #JOB_9_STEP_01) AND "Unit1.Em5.ControlNodes".transferPnPRight.sequence.status.seqActive AND "Unit1.Em5.ControlNodes".transferPnPRight."step".transition1[901],
                         PT := T#210ms);
   IF #statTonTime[901].Q THEN
       "Unit1.Em5.ControlNodes".transferPnPRight.sequence.status.nextStep := #JOB_9_STEP_10;
   END_IF;
END_REGION

